KUKA KRL program: EPS_2_251245_SANMH2A_A_20250910012814.src

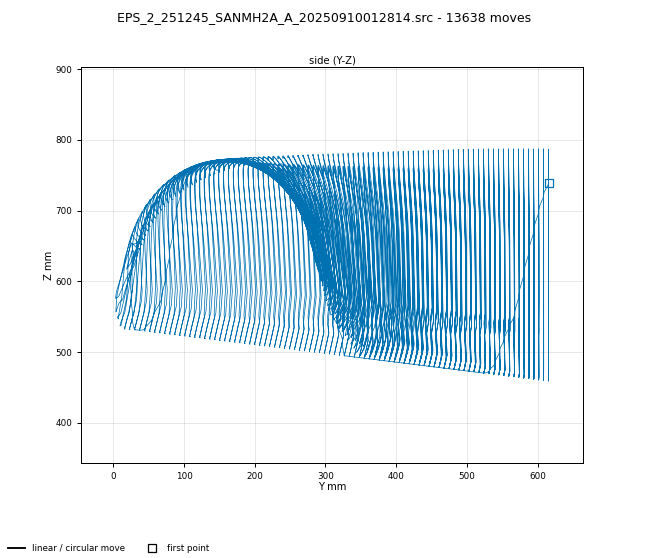
[picture p0: tool path of EPS_2_251245_SANMH2A_A_20250910012814.src, 13638 of 13640 moves have a stored position in this frame; points joined in program order, loops and branches not executed]
&ACCESS RVP
&REL 4
&COMMENT QRS 19112012
&PARAM EDITMASK = *
DEF PART()
EXT BAS (BAS_COMMAND :IN,REAL :IN )
INT I
BAS (#INITMOV,0 )

;KUKA QRS Post kuka4.cps  Date:22-06-2017 !

File_ID=2819

QRS_PRE_INIT()

;Init var - Until changes are made in qrs_pre_init
Outlet_Square_prg=0
Inlet_1_Square_prg=0
Inlet_2_Square_prg=0
Inlet_3_Square_prg=0
Inlet_4_Square_prg=0
Inlet_5_Square_prg=0

Outlet_1={X 0.000, Y 516.340, Z 662.000, B 0.000, E1 0.000 }
Inlet_1={X 0.000, Y 521.550, Z 654.000, B 0.000, E1 91.000 }
Inlet_2={X 0.000, Y 521.330, Z 657.000, B 0.000, E1 270.000 }
Outlet_1_type=251
Inlet_1_type=201
Inlet_2_type=201
;QRS#1=Sidecore dimensions
;QRS#2=250-10" PVC SDR 35
;QRS#3=200-8" PVC SDR 35
;QRS#4=200-8" PVC SDR 35
;QRS#5=
;QRS#6=
;QRS#7=
;QRS#8=
;QRS#9=14M PSX
;QRS#10=12-08 PSX
;QRS#11=12-08 PSX
;QRS#12=
;QRS#13=
;QRS#14=
;QRS#15=
;QRS#16=1220x127x1067 3,5'
;QRS#17=EPS Height
;QRS#18=787,5
;QRS#19=*
;QRS#20= UPDATED VERSION 22-06-2017
;QRS#21=*
Outlet_Square=0100
Inlet_1_Square=0100
Inlet_2_Square=0100
Inlet_3_Square=0
Inlet_4_Square=0
Inlet_5_Square=0
Mill_Square=1
Outlet_Square_Prg=205
Inlet_1_Square_prg=204
Inlet_2_Square_prg=204

QRS_INIT()

$ADVANCE=5

; T1
PTP {E1 173.419,E2 173.419}
PTP {X 0,Y 615.495,A -85,B 0,C 180,E1 173.419,E2 173.419,E3 0,E4 0,E5 0,E6 0}
QRS_SPEED_INIT()
LIN {X 0,Y 615.495,Z 739.089,A -85,B 0,C 180,E1 173.419,E2 173.419,E3 0,E4 0,E5 0,E6 0} C_VEL
LIN {X 0,Y 615.496,Z 732.969,A -85,B 0,C 180,E1 172.455,E2 172.455} C_VEL
LIN {X 0,Y 615.497,Z 725.117,A -85,B 0,C 180,E1 171.464,E2 171.464} C_VEL
LIN {X 0,Y 615.498,Z 715.327,A -85,B 0,C 180,E1 170.47,E2 170.47} C_VEL
LIN {X 0,Y 615.498,Z 705.048,A -85,B 0,C 180,E1 169.64,E2 169.64} C_VEL
LIN {X 0,Y 615.477,Z 693.364,A -85,B 0,C 180,E1 168.885,E2 168.885} C_VEL
LIN {X 0,Y 615.498,Z 681.888,A -85,B 0,C 180,E1 168.306,E2 168.306} C_VEL
LIN {X 0,Y 615.478,Z 669.89,A -85,B 0,C 180,E1 167.846,E2 167.846} C_VEL
LIN {X 0,Y 615.488,Z 657.742,A -85,B 0,C 180,E1 167.512,E2 167.512} C_VEL
LIN {X 0,Y 615.488,Z 644.369,A -85,B 0,C 180,E1 167.281,E2 167.281} C_VEL
LIN {X 0,Y 615.476,Z 541.661,A -85,B 0,C 180,E1 166.073,E2 166.073} C_VEL
LIN {X 0,Y 615.487,Z 518.802,A -85,B 0,C 180,E1 163.243,E2 163.243} C_VEL
LIN {X 0,Y 615.488,Z 495.468,A -85,B 0,C 180,E1 160.315,E2 160.315} C_VEL
LIN {X 0,Y 615.499,Z 472.639,A -85,B 0,C 180,E1 157.405,E2 157.405} C_VEL
LIN {X 0,Y 615.483,Z 458.809,A -85,B 0,C 180,E1 155.593,E2 155.593} C_VEL
LIN {X 0,Y 615.477,Z 458.815,A -85,B 0,C 180,E1 152.822,E2 152.822} C_VEL
LIN {X 0,Y 615.488,Z 458.822,A -85,B 0,C 180,E1 150.206,E2 150.206} C_VEL
LIN {X 0,Y 615.484,Z 458.808,A -85,B 0,C 180,E1 147.542,E2 147.542} C_VEL
LIN {X 0,Y 615.49,Z 458.807,A -85,B 0,C 180,E1 145.185,E2 145.185} C_VEL
LIN {X 0,Y 615.476,Z 458.818,A -85,B 0,C 180,E1 142.757,E2 142.757} C_VEL
LIN {X 0,Y 615.478,Z 458.815,A -85,B 0,C 180,E1 139.912,E2 139.912} C_VEL
LIN {X 0,Y 615.478,Z 458.81,A -85,B 0,C 180,E1 137.646,E2 137.646} C_VEL
LIN {X 0,Y 615.48,Z 458.814,A -85,B 0,C 180,E1 134.931,E2 134.931} C_VEL
LIN {X 0,Y 615.488,Z 458.816,A -85,B 0,C 180,E1 132.08,E2 132.08} C_VEL
LIN {X 0,Y 615.477,Z 458.812,A -85,B 0,C 180,E1 129.751,E2 129.751} C_VEL
LIN {X 0,Y 615.483,Z 458.813,A -85,B 0,C 180,E1 126.936,E2 126.936} C_VEL
LIN {X 0,Y 615.487,Z 458.814,A -85,B 0,C 180,E1 124.022,E2 124.022} C_VEL
LIN {X 0,Y 615.477,Z 458.81,A -85,B 0,C 180,E1 121.686,E2 121.686} C_VEL
LIN {X 0,Y 615.478,Z 458.809,A -85,B 0,C 180,E1 119.407,E2 119.407} C_VEL
LIN {X 0,Y 615.491,Z 458.81,A -85,B 0,C 180,E1 117.046,E2 117.046} C_VEL
LIN {X 0,Y 615.497,Z 458.818,A -85,B 0,C 180,E1 114.272,E2 114.272} C_VEL
LIN {X 0,Y 615.48,Z 458.809,A -85,B 0,C 180,E1 111.432,E2 111.432} C_VEL
LIN {X 0,Y 615.495,Z 458.822,A -85,B 0,C 180,E1 108.607,E2 108.607} C_VEL
LIN {X 0,Y 615.486,Z 458.811,A -85,B 0,C 180,E1 105.905,E2 105.905} C_VEL
LIN {X 0,Y 615.488,Z 458.809,A -85,B 0,C 180,E1 103.201,E2 103.201} C_VEL
LIN {X 0,Y 615.494,Z 458.826,A -85,B 0,C 180,E1 100.527,E2 100.527} C_VEL
LIN {X 0,Y 615.487,Z 458.81,A -85,B 0,C 180,E1 97.876,E2 97.876} C_VEL
LIN {X 0,Y 615.479,Z 458.811,A -85,B 0,C 180,E1 95.241,E2 95.241} C_VEL
LIN {X 0,Y 615.497,Z 458.823,A -85,B 0,C 180,E1 92.618,E2 92.618} C_VEL
LIN {X 0,Y 615.489,Z 458.811,A -85,B 0,C 180,E1 90,E2 90} C_VEL
LIN {X 0,Y 615.478,Z 458.81,A -85,B 0,C 180,E1 87.382,E2 87.382} C_VEL
LIN {X 0,Y 615.495,Z 458.819,A -85,B 0,C 180,E1 84.759,E2 84.759} C_VEL
LIN {X 0,Y 615.493,Z 458.812,A -85,B 0,C 180,E1 82.124,E2 82.124} C_VEL
LIN {X 0,Y 615.476,Z 458.81,A -85,B 0,C 180,E1 79.473,E2 79.473} C_VEL
LIN {X 0,Y 615.496,Z 458.818,A -85,B 0,C 180,E1 76.799,E2 76.799} C_VEL
LIN {X 0,Y 615.491,Z 458.811,A -85,B 0,C 180,E1 74.095,E2 74.095} C_VEL
LIN {X 0,Y 615.477,Z 458.811,A -85,B 0,C 180,E1 71.354,E2 71.354} C_VEL
LIN {X 0,Y 615.496,Z 458.824,A -85,B 0,C 180,E1 68.568,E2 68.568} C_VEL
LIN {X 0,Y 615.487,Z 458.807,A -85,B 0,C 180,E1 65.728,E2 65.728} C_VEL
LIN {X 0,Y 615.492,Z 458.82,A -85,B 0,C 180,E1 62.823,E2 62.823} C_VEL
LIN {X 0,Y 615.499,Z 458.805,A -85,B 0,C 180,E1 59.84,E2 59.84} C_VEL
LIN {X 0,Y 615.481,Z 458.809,A -85,B 0,C 180,E1 57.542,E2 57.542} C_VEL
LIN {X 0,Y 615.478,Z 458.814,A -85,B 0,C 180,E1 55.184,E2 55.184} C_VEL
LIN {X 0,Y 615.494,Z 458.823,A -85,B 0,C 180,E1 52.758,E2 52.758} C_VEL
LIN {X 0,Y 615.491,Z 458.807,A -85,B 0,C 180,E1 49.911,E2 49.911} C_VEL
LIN {X 0,Y 615.49,Z 458.806,A -85,B 0,C 180,E1 47.647,E2 47.647} C_VEL
LIN {X 0,Y 615.481,Z 458.821,A -85,B 0,C 180,E1 44.931,E2 44.931} C_VEL
LIN {X 0,Y 615.478,Z 458.812,A -85,B 0,C 180,E1 42.079,E2 42.079} C_VEL
LIN {X 0,Y 615.498,Z 458.805,A -85,B 0,C 180,E1 39.749,E2 39.749} C_VEL
LIN {X 0,Y 615.478,Z 458.822,A -85,B 0,C 180,E1 36.935,E2 36.935} C_VEL
LIN {X 0,Y 615.491,Z 458.826,A -85,B 0,C 180,E1 34.701,E2 34.701} C_VEL
LIN {X 0,Y 615.479,Z 458.816,A -85,B 0,C 180,E1 32.329,E2 32.329} C_VEL
LIN {X 0,Y 615.488,Z 458.807,A -85,B 0,C 180,E1 29.794,E2 29.794} C_VEL
LIN {X 0,Y 615.482,Z 458.819,A -85,B 0,C 180,E1 27.043,E2 27.043} C_VEL
LIN {X 0,Y 615.478,Z 458.815,A -85,B 0,C 180,E1 24.272,E2 24.272} C_VEL
LIN {X 0,Y 615.486,Z 458.917,A -85,B 0,C 180,E1 23.49,E2 23.49} C_VEL
LIN {X 0,Y 615.485,Z 480.604,A -85,B 0,C 180,E1 20.731,E2 20.731} C_VEL
LIN {X 0,Y 615.49,Z 502.793,A -85,B 0,C 180,E1 17.957,E2 17.957} C_VEL
LIN {X 0,Y 615.491,Z 524.956,A -85,B 0,C 180,E1 15.226,E2 15.226} C_VEL
LIN {X 0,Y 615.481,Z 544.498,A -85,B 0,C 180,E1 12.845,E2 12.845} C_VEL
LIN {X 0,Y 615.489,Z 653.144,A -85,B 0,C 180,E1 11.548,E2 11.548} C_VEL
LIN {X 0,Y 615.484,Z 665.724,A -85,B 0,C 180,E1 11.277,E2 11.277} C_VEL
LIN {X 0,Y 615.49,Z 679.129,A -85,B 0,C 180,E1 10.841,E2 10.841} C_VEL
LIN {X 0,Y 615.481,Z 691.697,A -85,B 0,C 180,E1 10.278,E2 10.278} C_VEL
LIN {X 0,Y 615.493,Z 703.076,A -85,B 0,C 180,E1 9.613,E2 9.613} C_VEL
LIN {X 0,Y 615.498,Z 713.323,A -85,B 0,C 180,E1 8.867,E2 8.867} C_VEL
LIN {X 0,Y 615.498,Z 722.534,A -85,B 0,C 180,E1 8.041,E2 8.041} C_VEL
LIN {X 0,Y 615.499,Z 731.392,A -85,B 0,C 180,E1 7.057,E2 7.057} C_VEL
LIN {X 0,Y 615.497,Z 738.623,A -85,B 0,C 180,E1 6.063,E2 6.063} C_VEL
LIN {X 0,Y 615.497,Z 743.458,A -85,B 0,C 180,E1 5.241,E2 5.241} C_VEL
LIN {X 0,Y 615.493,Z 748.158,A -85,B 0,C 180,E1 4.256,E2 4.256} C_VEL
LIN {X 0,Y 615.495,Z 751.754,A -85,B 0,C 180,E1 3.273,E2 3.273} C_VEL
LIN {X 0,Y 615.496,Z 753.615,A -85,B 0,C 180,E1 2.618,E2 2.618} C_VEL
LIN {X 0,Y 615.497,Z 755.034,A -85,B 0,C 180,E1 1.963,E2 1.963} C_VEL
LIN {X 0,Y 615.496,Z 756.642,A -85,B 0,C 180,E1 0.654,E2 0.654} C_VEL
LIN {X 0,Y 615.494,Z 756.884,A -85,B 0,C 180,E1 0,E2 0} C_VEL
LIN {X 0,Y 615.496,Z 756.705,A -85,B 0,C 180,E1 -0.654,E2 -0.654} C_VEL
LIN {X 0,Y 615.496,Z 755.183,A -85,B 0,C 180,E1 -1.963,E2 -1.963} C_VEL
LIN {X 0,Y 615.498,Z 753.841,A -85,B 0,C 180,E1 -2.618,E2 -2.618} C_VEL
LIN {X 0,Y 615.496,Z 750.994,A -85,B 0,C 180,E1 -3.601,E2 -3.601} C_VEL
LIN {X 0,Y 615.499,Z 747.134,A -85,B 0,C 180,E1 -4.584,E2 -4.584} C_VEL
LIN {X 0,Y 615.498,Z 742.151,A -85,B 0,C 180,E1 -5.57,E2 -5.57} C_VEL
LIN {X 0,Y 615.497,Z 735.701,A -85,B 0,C 180,E1 -6.583,E2 -6.583} C_VEL
LIN {X 0,Y 615.497,Z 728.036,A -85,B 0,C 180,E1 -7.545,E2 -7.545} C_VEL
LIN {X 0,Y 615.498,Z 718.258,A -85,B 0,C 180,E1 -8.537,E2 -8.537} C_VEL
LIN {X 0,Y 615.497,Z 707.993,A -85,B 0,C 180,E1 -9.364,E2 -9.364} C_VEL
LIN {X 0,Y 615.476,Z 696.432,A -85,B 0,C 180,E1 -10.112,E2 -10.112} C_VEL
LIN {X 0,Y 615.497,Z 684.578,A -85,B 0,C 180,E1 -10.707,E2 -10.707} C_VEL
LIN {X 0,Y 615.478,Z 671.66,A -85,B 0,C 180,E1 -11.193,E2 -11.193} C_VEL
LIN {X 0,Y 615.486,Z 659.058,A -85,B 0,C 180,E1 -11.527,E2 -11.527} C_VEL
LIN {X 0,Y 615.487,Z 645.933,A -85,B 0,C 180,E1 -11.736,E2 -11.736} C_VEL
LIN {X 0,Y 615.478,Z 544.549,A -85,B 0,C 180,E1 -12.929,E2 -12.929} C_VEL
LIN {X 0,Y 615.488,Z 521.533,A -85,B 0,C 180,E1 -15.735,E2 -15.735} C_VEL
LIN {X 0,Y 615.491,Z 497.97,A -85,B 0,C 180,E1 -18.646,E2 -18.646} C_VEL
LIN {X 0,Y 615.497,Z 475.763,A -85,B 0,C 180,E1 -21.432,E2 -21.432} C_VEL
LIN {X 0,Y 615.486,Z 458.809,A -85,B 0,C 180,E1 -23.612,E2 -23.612} C_VEL
LIN {X 0,Y 615.48,Z 458.818,A -85,B 0,C 180,E1 -26.445,E2 -26.445} C_VEL
LIN {X 0,Y 615.49,Z 458.823,A -85,B 0,C 180,E1 -28.658,E2 -28.658} C_VEL
LIN {X 0,Y 615.477,Z 458.818,A -85,B 0,C 180,E1 -31.084,E2 -31.084} C_VEL
LIN {X 0,Y 615.485,Z 458.808,A -85,B 0,C 180,E1 -33.533,E2 -33.533} C_VEL
LIN {X 0,Y 615.484,Z 458.82,A -85,B 0,C 180,E1 -36.425,E2 -36.425} C_VEL
LIN {X 0,Y 615.479,Z 458.816,A -85,B 0,C 180,E1 -39.061,E2 -39.061} C_VEL
LIN {X 0,Y 615.482,Z 458.809,A -85,B 0,C 180,E1 -41.474,E2 -41.474} C_VEL
LIN {X 0,Y 615.479,Z 458.817,A -85,B 0,C 180,E1 -44.15,E2 -44.15} C_VEL
LIN {X 0,Y 615.485,Z 458.814,A -85,B 0,C 180,E1 -46.953,E2 -46.953} C_VEL
LIN {X 0,Y 615.478,Z 458.81,A -85,B 0,C 180,E1 -49.393,E2 -49.393} C_VEL
LIN {X 0,Y 615.492,Z 458.813,A -85,B 0,C 180,E1 -51.988,E2 -51.988} C_VEL
LIN {X 0,Y 615.497,Z 458.825,A -85,B 0,C 180,E1 -54.385,E2 -54.385} C_VEL
LIN {X 0,Y 615.49,Z 458.814,A -85,B 0,C 180,E1 -56.764,E2 -56.764} C_VEL
LIN {X 0,Y 615.478,Z 458.811,A -85,B 0,C 180,E1 -59.08,E2 -59.08} C_VEL
LIN {X 0,Y 615.481,Z 458.81,A -85,B 0,C 180,E1 -61.551,E2 -61.551} C_VEL
LIN {X 0,Y 615.493,Z 458.82,A -85,B 0,C 180,E1 -64.43,E2 -64.43} C_VEL
LIN {X 0,Y 615.48,Z 458.809,A -85,B 0,C 180,E1 -67.155,E2 -67.155} C_VEL
LIN {X 0,Y 615.475,Z 458.897,A -85,B 0,C 180,E1 -67.374,E2 -67.374} C_VEL
LIN {X 0,Y 615.496,Z 484.108,A -85,B 0,C 180,E1 -70.141,E2 -70.141} C_VEL
LIN {X 0,Y 615.495,Z 511.278,A -85,B 0,C 180,E1 -73.072,E2 -73.072} C_VEL
LIN {X 0,Y 615.488,Z 523.651,A -85,B 0,C 180,E1 -74.392,E2 -74.392} C_VEL
LIN {X 0,Y 615.485,Z 662.162,A -85,B 0,C 180,E1 -76.05,E2 -76.05} C_VEL
LIN {X 0,Y 615.486,Z 675.855,A -85,B 0,C 180,E1 -76.336,E2 -76.336} C_VEL
LIN {X 0,Y 615.496,Z 689.566,A -85,B 0,C 180,E1 -76.757,E2 -76.757} C_VEL
LIN {X 0,Y 615.497,Z 702.836,A -85,B 0,C 180,E1 -77.302,E2 -77.302} C_VEL
LIN {X 0,Y 615.492,Z 715.599,A -85,B 0,C 180,E1 -77.972,E2 -77.972} C_VEL
LIN {X 0,Y 615.499,Z 727.182,A -85,B 0,C 180,E1 -78.724,E2 -78.724} C_VEL
LIN {X 0,Y 615.498,Z 738.748,A -85,B 0,C 180,E1 -79.64,E2 -79.64} C_VEL
LIN {X 0,Y 615.497,Z 749.088,A -85,B 0,C 180,E1 -80.636,E2 -80.636} C_VEL
LIN {X 0,Y 615.497,Z 757.602,A -85,B 0,C 180,E1 -81.629,E2 -81.629} C_VEL
LIN {X 0,Y 615.496,Z 765.726,A -85,B 0,C 180,E1 -82.784,E2 -82.784} C_VEL
LIN {X 0,Y 615.496,Z 771.43,A -85,B 0,C 180,E1 -83.773,E2 -83.773} C_VEL
LIN {X 0,Y 615.495,Z 776.08,A -85,B 0,C 180,E1 -84.759,E2 -84.759} C_VEL
LIN {X 0,Y 615.494,Z 780.902,A -85,B 0,C 180,E1 -86.072,E2 -86.072} C_VEL
LIN {X 0,Y 615.496,Z 784.252,A -85,B 0,C 180,E1 -87.382,E2 -87.382} C_VEL
LIN {X 0,Y 615.489,Z 786.229,A -85,B 0,C 180,E1 -88.691,E2 -88.691} C_VEL
LIN {X 0,Y 615.493,Z 786.889,A -85,B 0,C 180,E1 -90,E2 -90} C_VEL
LIN {X 0,Y 615.489,Z 786.229,A -85,B 0,C 180,E1 -91.309,E2 -91.309} C_VEL
LIN {X 0,Y 615.496,Z 784.252,A -85,B 0,C 180,E1 -92.618,E2 -92.618} C_VEL
LIN {X 0,Y 615.494,Z 780.901,A -85,B 0,C 180,E1 -93.929,E2 -93.929} C_VEL
LIN {X 0,Y 615.495,Z 776.08,A -85,B 0,C 180,E1 -95.241,E2 -95.241} C_VEL
LIN {X 0,Y 615.495,Z 769.628,A -85,B 0,C 180,E1 -96.557,E2 -96.557} C_VEL
LIN {X 0,Y 615.497,Z 762.44,A -85,B 0,C 180,E1 -97.711,E2 -97.711} C_VEL
LIN {X 0,Y 615.497,Z 754.902,A -85,B 0,C 180,E1 -98.702,E2 -98.702} C_VEL
LIN {X 0,Y 615.495,Z 745.852,A -85,B 0,C 180,E1 -99.696,E2 -99.696} C_VEL
LIN {X 0,Y 615.497,Z 735.756,A -85,B 0,C 180,E1 -100.618,E2 -100.618} C_VEL
LIN {X 0,Y 615.498,Z 724.855,A -85,B 0,C 180,E1 -101.443,E2 -101.443} C_VEL
LIN {X 0,Y 615.488,Z 712.703,A -85,B 0,C 180,E1 -102.195,E2 -102.195} C_VEL
LIN {X 0,Y 615.495,Z 699.087,A -85,B 0,C 180,E1 -102.865,E2 -102.865} C_VEL
LIN {X 0,Y 615.492,Z 685.829,A -85,B 0,C 180,E1 -103.369,E2 -103.369} C_VEL
LIN {X 0,Y 615.484,Z 672.279,A -85,B 0,C 180,E1 -103.748,E2 -103.748} C_VEL
LIN {X 0,Y 615.486,Z 658.082,A -85,B 0,C 180,E1 -104.008,E2 -104.008} C_VEL
LIN {X 0,Y 615.488,Z 523.65,A -85,B 0,C 180,E1 -105.608,E2 -105.608} C_VEL
LIN {X 0,Y 615.488,Z 497.182,A -85,B 0,C 180,E1 -108.443,E2 -108.443} C_VEL
LIN {X 0,Y 615.493,Z 471.313,A -85,B 0,C 180,E1 -111.256,E2 -111.256} C_VEL
LIN {X 0,Y 615.475,Z 458.811,A -85,B 0,C 180,E1 -112.657,E2 -112.657} C_VEL
LIN {X 0,Y 615.488,Z 458.809,A -85,B 0,C 180,E1 -114.992,E2 -114.992} C_VEL
LIN {X 0,Y 615.492,Z 458.817,A -85,B 0,C 180,E1 -117.915,E2 -117.915} C_VEL
LIN {X 0,Y 615.499,Z 458.808,A -85,B 0,C 180,E1 -120.16,E2 -120.16} C_VEL
LIN {X 0,Y 615.481,Z 458.809,A -85,B 0,C 180,E1 -122.458,E2 -122.458} C_VEL
LIN {X 0,Y 615.478,Z 458.813,A -85,B 0,C 180,E1 -124.816,E2 -124.816} C_VEL
LIN {X 0,Y 615.492,Z 458.823,A -85,B 0,C 180,E1 -127.242,E2 -127.242} C_VEL
LIN {X 0,Y 615.489,Z 458.808,A -85,B 0,C 180,E1 -130.089,E2 -130.089} C_VEL
LIN {X 0,Y 615.486,Z 458.823,A -85,B 0,C 180,E1 -133.047,E2 -133.047} C_VEL
LIN {X 0,Y 615.482,Z 458.809,A -85,B 0,C 180,E1 -136.003,E2 -136.003} C_VEL
LIN {X 0,Y 615.49,Z 458.823,A -85,B 0,C 180,E1 -138.906,E2 -138.906} C_VEL
LIN {X 0,Y 615.496,Z 458.82,A -85,B 0,C 180,E1 -141.096,E2 -141.096} C_VEL
LIN {X 0,Y 615.481,Z 458.811,A -85,B 0,C 180,E1 -143.575,E2 -143.575} C_VEL
LIN {X 0,Y 615.479,Z 458.81,A -85,B 0,C 180,E1 -145.977,E2 -145.977} C_VEL
LIN {X 0,Y 615.493,Z 458.82,A -85,B 0,C 180,E1 -148.914,E2 -148.914} C_VEL
LIN {X 0,Y 615.484,Z 458.809,A -85,B 0,C 180,E1 -151.551,E2 -151.551} C_VEL
LIN {X 0,Y 615.499,Z 458.821,A -85,B 0,C 180,E1 -154.43,E2 -154.43} C_VEL
LIN {X 0,Y 615.484,Z 458.811,A -85,B 0,C 180,E1 -157.155,E2 -157.155} C_VEL
LIN {X 0,Y 615.479,Z 458.836,A -85,B 0,C 180,E1 -157.708,E2 -157.708} C_VEL
LIN {X 0,Y 615.492,Z 480.389,A -85,B 0,C 180,E1 -160.489,E2 -160.489} C_VEL
LIN {X 0,Y 615.492,Z 503.466,A -85,B 0,C 180,E1 -163.413,E2 -163.413} C_VEL
LIN {X 0,Y 615.485,Z 526.538,A -85,B 0,C 180,E1 -166.294,E2 -166.294} C_VEL
LIN {X 0,Y 615.48,Z 541.632,A -85,B 0,C 180,E1 -168.16,E2 -168.16} C_VEL
LIN {X 0,Y 615.491,Z 651.28,A -85,B 0,C 180,E1 -169.473,E2 -169.473} C_VEL
LIN {X 0,Y 615.484,Z 664.198,A -85,B 0,C 180,E1 -169.764,E2 -169.764} C_VEL
LIN {X 0,Y 615.49,Z 676.689,A -85,B 0,C 180,E1 -170.179,E2 -170.179} C_VEL
LIN {X 0,Y 615.482,Z 688.618,A -85,B 0,C 180,E1 -170.718,E2 -170.718} C_VEL
LIN {X 0,Y 615.494,Z 699.982,A -85,B 0,C 180,E1 -171.381,E2 -171.381} C_VEL
LIN {X 0,Y 615.498,Z 710.219,A -85,B 0,C 180,E1 -172.124,E2 -172.124} C_VEL
LIN {X 0,Y 615.499,Z 719.371,A -85,B 0,C 180,E1 -172.943,E2 -172.943} C_VEL
LIN {X 0,Y 615.496,Z 728.347,A -85,B 0,C 180,E1 -173.937,E2 -173.937} C_VEL
LIN {X 0,Y 615.497,Z 735.529,A -85,B 0,C 180,E1 -174.923,E2 -174.923} C_VEL
LIN {X 0,Y 615.493,Z 740.375,A -85,B 0,C 180,E1 -175.744,E2 -175.744} C_VEL
LIN {X 0,Y 615.496,Z 745.086,A -85,B 0,C 180,E1 -176.727,E2 -176.727} C_VEL
LIN {X 0,Y 615.498,Z 748.698,A -85,B 0,C 180,E1 -177.71,E2 -177.71} C_VEL
LIN {X 0,Y 615.496,Z 751.317,A -85,B 0,C 180,E1 -178.691,E2 -178.691} C_VEL
LIN {X 0,Y 615.495,Z 753.389,A -85,B 0,C 180,E1 -180,E2 -180} C_VEL
LIN {X 0,Y 615.496,Z 753.831,A -85,B 0,C 180,E1 -181.309,E2 -181.309} C_VEL
LIN {X 0,Y 615.495,Z 752.757,A -85,B 0,C 180,E1 -182.618,E2 -182.618} C_VEL
LIN {X 0,Y 615.497,Z 751.59,A -85,B 0,C 180,E1 -183.273,E2 -183.273} C_VEL
LIN {X 0,Y 615.494,Z 750.023,A -85,B 0,C 180,E1 -183.928,E2 -183.928} C_VEL
LIN {X 0,Y 615.494,Z 746.868,A -85,B 0,C 180,E1 -184.913,E2 -184.913} C_VEL
LIN {X 0,Y 615.498,Z 742.661,A -85,B 0,C 180,E1 -185.898,E2 -185.898} C_VEL
LIN {X 0,Y 615.495,Z 739.089,A -85,B 0,C 180,E1 -186.581,E2 -186.581} C_VEL
LIN {X 0,Y 614.823,Z 736.384,A -85,B 0,C 180,E1 -187.059,E2 -187.059} C_VEL
LIN {X 0,Y 611.979,Z 731.579,A -85,B 0,C 180,E1 -187.825,E2 -187.825} C_VEL
LIN {X 0,Y 609.133,Z 726.046,A -85,B 0,C 180,E1 -188.558,E2 -188.558} C_VEL
LIN {X 0,Y 608.473,Z 722.206,A -85,B 0,C 180,E1 -188.982,E2 -188.982} C_VEL
LIN {X 0,Y 608.488,Z 713.552,A -85,B 0,C 180,E1 -189.809,E2 -189.809} C_VEL
LIN {X 0,Y 608.492,Z 702.773,A -85,B 0,C 180,E1 -190.649,E2 -190.649} C_VEL
LIN {X 0,Y 608.481,Z 691.914,A -85,B 0,C 180,E1 -191.324,E2 -191.324} C_VEL
LIN {X 0,Y 608.508,Z 679.767,A -85,B 0,C 180,E1 -191.914,E2 -191.914} C_VEL
LIN {X 0,Y 608.523,Z 667.028,A -85,B 0,C 180,E1 -192.379,E2 -192.379} C_VEL
LIN {X 0,Y 608.553,Z 654.338,A -85,B 0,C 180,E1 -192.696,E2 -192.696} C_VEL
LIN {X 0,Y 608.536,Z 638.078,A -85,B 0,C 180,E1 -192.93,E2 -192.93} C_VEL
LIN {X 0,Y 608.466,Z 541.843,A -85,B 0,C 180,E1 -194.072,E2 -194.072} C_VEL
LIN {X 0,Y 608.495,Z 520.137,A -85,B 0,C 180,E1 -196.783,E2 -196.783} C_VEL
LIN {X 0,Y 608.555,Z 498.132,A -85,B 0,C 180,E1 -199.567,E2 -199.567} C_VEL
LIN {X 0,Y 608.592,Z 475.299,A -85,B 0,C 180,E1 -202.506,E2 -202.506} C_VEL
LIN {X 0,Y 608.482,Z 459.811,A -85,B 0,C 180,E1 -204.538,E2 -204.538} C_VEL
LIN {X 0,Y 608.473,Z 459.814,A -85,B 0,C 180,E1 -207.206,E2 -207.206} C_VEL
LIN {X 0,Y 608.466,Z 459.816,A -85,B 0,C 180,E1 -209.971,E2 -209.971} C_VEL
LIN {X 0,Y 608.452,Z 459.813,A -85,B 0,C 180,E1 -212.88,E2 -212.88} C_VEL
LIN {X 0,Y 608.452,Z 459.817,A -85,B 0,C 180,E1 -215.277,E2 -215.277} C_VEL
LIN {X 0,Y 608.461,Z 459.819,A -85,B 0,C 180,E1 -217.747,E2 -217.747} C_VEL
LIN {X 0,Y 608.446,Z 459.814,A -85,B 0,C 180,E1 -220.328,E2 -220.328} C_VEL
LIN {X 0,Y 608.469,Z 459.816,A -85,B 0,C 180,E1 -223.308,E2 -223.308} C_VEL
LIN {X 0,Y 608.47,Z 459.812,A -85,B 0,C 180,E1 -226.13,E2 -226.13} C_VEL
LIN {X 0,Y 608.453,Z 459.813,A -85,B 0,C 180,E1 -228.823,E2 -228.823} C_VEL
LIN {X 0,Y 608.469,Z 459.817,A -85,B 0,C 180,E1 -231.76,E2 -231.76} C_VEL
LIN {X 0,Y 608.447,Z 459.817,A -85,B 0,C 180,E1 -233.955,E2 -233.955} C_VEL
LIN {X 0,Y 608.449,Z 459.813,A -85,B 0,C 180,E1 -236.328,E2 -236.328} C_VEL
LIN {X 0,Y 608.449,Z 459.813,A -85,B 0,C 180,E1 -238.732,E2 -238.732} C_VEL
LIN {X 0,Y 608.477,Z 459.817,A -85,B 0,C 180,E1 -241.379,E2 -241.379} C_VEL
LIN {X 0,Y 608.444,Z 459.817,A -85,B 0,C 180,E1 -243.964,E2 -243.964} C_VEL
LIN {X 0,Y 608.466,Z 459.812,A -85,B 0,C 180,E1 -246.155,E2 -246.155} C_VEL
LIN {X 0,Y 608.469,Z 459.81,A -85,B 0,C 180,E1 -248.308,E2 -248.308} C_VEL
LIN {X 0,Y 608.477,Z 459.816,A -85,B 0,C 180,E1 -251.283,E2 -251.283} C_VEL
LIN {X 0,Y 608.464,Z 459.815,A -85,B 0,C 180,E1 -253.906,E2 -253.906} C_VEL
LIN {X 0,Y 608.465,Z 459.811,A -85,B 0,C 180,E1 -256.643,E2 -256.643} C_VEL
LIN {X 0,Y 608.472,Z 459.818,A -85,B 0,C 180,E1 -259.35,E2 -259.35} C_VEL
LIN {X 0,Y 608.48,Z 459.811,A -85,B 0,C 180,E1 -262.033,E2 -262.033} C_VEL
LIN {X 0,Y 608.46,Z 459.812,A -85,B 0,C 180,E1 -264.698,E2 -264.698} C_VEL
LIN {X 0,Y 608.487,Z 459.817,A -85,B 0,C 180,E1 -267.352,E2 -267.352} C_VEL
LIN {X 0,Y 608.48,Z 459.811,A -85,B 0,C 180,E1 -270,E2 -270} C_VEL
LIN {X 0,Y 608.47,Z 459.81,A -85,B 0,C 180,E1 -272.648,E2 -272.648} C_VEL
LIN {X 0,Y 608.474,Z 459.818,A -85,B 0,C 180,E1 -275.302,E2 -275.302} C_VEL
LIN {X 0,Y 608.481,Z 459.811,A -85,B 0,C 180,E1 -277.967,E2 -277.967} C_VEL
LIN {X 0,Y 608.458,Z 459.812,A -85,B 0,C 180,E1 -280.65,E2 -280.65} C_VEL
LIN {X 0,Y 608.472,Z 459.82,A -85,B 0,C 180,E1 -283.356,E2 -283.356} C_VEL
LIN {X 0,Y 608.462,Z 459.812,A -85,B 0,C 180,E1 -286.094,E2 -286.094} C_VEL
LIN {X 0,Y 608.455,Z 459.814,A -85,B 0,C 180,E1 -288.87,E2 -288.87} C_VEL
LIN {X 0,Y 608.477,Z 459.814,A -85,B 0,C 180,E1 -291.691,E2 -291.691} C_VEL
LIN {X 0,Y 608.455,Z 459.812,A -85,B 0,C 180,E1 -294.571,E2 -294.571} C_VEL
LIN {X 0,Y 608.485,Z 459.816,A -85,B 0,C 180,E1 -297.208,E2 -297.208} C_VEL
LIN {X 0,Y 608.471,Z 459.811,A -85,B 0,C 180,E1 -299.972,E2 -299.972} C_VEL
LIN {X 0,Y 608.459,Z 459.814,A -85,B 0,C 180,E1 -302.88,E2 -302.88} C_VEL
LIN {X 0,Y 608.44,Z 459.824,A -85,B 0,C 180,E1 -305.278,E2 -305.278} C_VEL
LIN {X 0,Y 608.473,Z 459.813,A -85,B 0,C 180,E1 -307.746,E2 -307.746} C_VEL
LIN {X 0,Y 608.451,Z 459.812,A -85,B 0,C 180,E1 -310.329,E2 -310.329} C_VEL
LIN {X 0,Y 608.486,Z 459.819,A -85,B 0,C 180,E1 -313.31,E2 -313.31} C_VEL
LIN {X 0,Y 608.468,Z 459.81,A -85,B 0,C 180,E1 -316.13,E2 -316.13} C_VEL
LIN {X 0,Y 608.449,Z 459.816,A -85,B 0,C 180,E1 -318.823,E2 -318.823} C_VEL
LIN {X 0,Y 608.466,Z 459.819,A -85,B 0,C 180,E1 -321.412,E2 -321.412} C_VEL
LIN {X 0,Y 608.449,Z 459.814,A -85,B 0,C 180,E1 -323.955,E2 -323.955} C_VEL
LIN {X 0,Y 608.451,Z 459.812,A -85,B 0,C 180,E1 -326.328,E2 -326.328} C_VEL
LIN {X 0,Y 608.447,Z 459.815,A -85,B 0,C 180,E1 -328.733,E2 -328.733} C_VEL
LIN {X 0,Y 608.475,Z 459.818,A -85,B 0,C 180,E1 -331.38,E2 -331.38} C_VEL
LIN {X 0,Y 608.478,Z 459.809,A -85,B 0,C 180,E1 -334.278,E2 -334.278} C_VEL
LIN {X 0,Y 608.504,Z 459.962,A -85,B 0,C 180,E1 -336.36,E2 -336.36} C_VEL
LIN {X 0,Y 608.596,Z 476.445,A -85,B 0,C 180,E1 -338.491,E2 -338.491} C_VEL
LIN {X 0,Y 608.545,Z 498.307,A -85,B 0,C 180,E1 -341.264,E2 -341.264} C_VEL
LIN {X 0,Y 608.519,Z 520.864,A -85,B 0,C 180,E1 -344.08,E2 -344.08} C_VEL
LIN {X 0,Y 608.473,Z 543.075,A -85,B 0,C 180,E1 -346.814,E2 -346.814} C_VEL
LIN {X 0,Y 608.481,Z 544.724,A -85,B 0,C 180,E1 -347.016,E2 -347.016} C_VEL
LIN {X 0,Y 608.554,Z 653.284,A -85,B 0,C 180,E1 -348.319,E2 -348.319} C_VEL
LIN {X 0,Y 608.531,Z 666.622,A -85,B 0,C 180,E1 -348.614,E2 -348.614} C_VEL
LIN {X 0,Y 608.511,Z 679.096,A -85,B 0,C 180,E1 -349.026,E2 -349.026} C_VEL
LIN {X 0,Y 608.509,Z 690.233,A -85,B 0,C 180,E1 -349.519,E2 -349.519} C_VEL
LIN {X 0,Y 608.488,Z 702.014,A -85,B 0,C 180,E1 -350.191,E2 -350.191} C_VEL
LIN {X 0,Y 608.474,Z 713.585,A -85,B 0,C 180,E1 -351.029,E2 -351.029} C_VEL
LIN {X 0,Y 608.464,Z 722.849,A -85,B 0,C 180,E1 -351.866,E2 -351.866} C_VEL
LIN {X 0,Y 608.466,Z 731.823,A -85,B 0,C 180,E1 -352.867,E2 -352.867} C_VEL
LIN {X 0,Y 608.444,Z 739.056,A -85,B 0,C 180,E1 -353.867,E2 -353.867} C_VEL
LIN {X 0,Y 608.462,Z 743.935,A -85,B 0,C 180,E1 -354.698,E2 -354.698} C_VEL
LIN {X 0,Y 608.439,Z 748.679,A -85,B 0,C 180,E1 -355.694,E2 -355.694} C_VEL
LIN {X 0,Y 608.426,Z 752.313,A -85,B 0,C 180,E1 -356.689,E2 -356.689} C_VEL
LIN {X 0,Y 608.425,Z 754.19,A -85,B 0,C 180,E1 -357.352,E2 -357.352} C_VEL
LIN {X 0,Y 608.442,Z 755.626,A -85,B 0,C 180,E1 -358.014,E2 -358.014} C_VEL
LIN {X 0,Y 608.439,Z 757.252,A -85,B 0,C 180,E1 -359.338,E2 -359.338} C_VEL
LIN {X 0,Y 608.434,Z 757.495,A -85,B 0,C 180,E1 -360,E2 -360} C_VEL
LIN {X 0,Y 608.439,Z 757.315,A -85,B 0,C 180,E1 -360.662,E2 -360.662} C_VEL
LIN {X 0,Y 608.441,Z 755.776,A -85,B 0,C 180,E1 -361.986,E2 -361.986} C_VEL
LIN {X 0,Y 608.426,Z 754.419,A -85,B 0,C 180,E1 -362.648,E2 -362.648} C_VEL
LIN {X 0,Y 608.449,Z 751.542,A -85,B 0,C 180,E1 -363.642,E2 -363.642} C_VEL
LIN {X 0,Y 608.433,Z 747.643,A -85,B 0,C 180,E1 -364.638,E2 -364.638} C_VEL
LIN {X 0,Y 608.449,Z 742.613,A -85,B 0,C 180,E1 -365.634,E2 -365.634} C_VEL
LIN {X 0,Y 608.442,Z 736.292,A -85,B 0,C 180,E1 -366.633,E2 -366.633} C_VEL
LIN {X 0,Y 608.475,Z 728.379,A -85,B 0,C 180,E1 -367.633,E2 -367.633} C_VEL
LIN {X 0,Y 608.472,Z 718.536,A -85,B 0,C 180,E1 -368.636,E2 -368.636} C_VEL
LIN {X 0,Y 608.48,Z 708.209,A -85,B 0,C 180,E1 -369.473,E2 -369.473} C_VEL
LIN {X 0,Y 608.473,Z 696.595,A -85,B 0,C 180,E1 -370.229,E2 -370.229} C_VEL
LIN {X 0,Y 608.525,Z 685.402,A -85,B 0,C 180,E1 -370.801,E2 -370.801} C_VEL
LIN {X 0,Y 608.527,Z 672.754,A -85,B 0,C 180,E1 -371.29,E2 -371.29} C_VEL
LIN {X 0,Y 608.53,Z 660.049,A -85,B 0,C 180,E1 -371.639,E2 -371.639} C_VEL
LIN {X 0,Y 608.559,Z 647.787,A -85,B 0,C 180,E1 -371.85,E2 -371.85} C_VEL
LIN {X 0,Y 608.466,Z 544.678,A -85,B 0,C 180,E1 -373.08,E2 -373.08} C_VEL
LIN {X 0,Y 608.497,Z 522.979,A -85,B 0,C 180,E1 -375.749,E2 -375.749} C_VEL
LIN {X 0,Y 608.56,Z 500.92,A -85,B 0,C 180,E1 -378.497,E2 -378.497} C_VEL
LIN {X 0,Y 608.564,Z 479.925,A -85,B 0,C 180,E1 -381.155,E2 -381.155} C_VEL
LIN {X 0,Y 608.6,Z 460.481,A -85,B 0,C 180,E1 -383.659,E2 -383.659} C_VEL
LIN {X 0,Y 608.485,Z 459.81,A -85,B 0,C 180,E1 -383.754,E2 -383.754} C_VEL
LIN {X 0,Y 608.447,Z 459.814,A -85,B 0,C 180,E1 -386.035,E2 -386.035} C_VEL
LIN {X 0,Y 608.473,Z 459.818,A -85,B 0,C 180,E1 -388.619,E2 -388.619} C_VEL
LIN {X 0,Y 608.447,Z 459.815,A -85,B 0,C 180,E1 -391.318,E2 -391.318} C_VEL
LIN {X 0,Y 608.475,Z 459.81,A -85,B 0,C 180,E1 -393.735,E2 -393.735} C_VEL
LIN {X 0,Y 608.449,Z 459.815,A -85,B 0,C 180,E1 -396.092,E2 -396.092} C_VEL
LIN {X 0,Y 608.467,Z 459.821,A -85,B 0,C 180,E1 -398.588,E2 -398.588} C_VEL
LIN {X 0,Y 608.457,Z 459.812,A -85,B 0,C 180,E1 -401.341,E2 -401.341} C_VEL
LIN {X 0,Y 608.45,Z 459.818,A -85,B 0,C 180,E1 -404.263,E2 -404.263} C_VEL
LIN {X 0,Y 608.453,Z 459.815,A -85,B 0,C 180,E1 -407.04,E2 -407.04} C_VEL
LIN {X 0,Y 608.455,Z 459.813,A -85,B 0,C 180,E1 -409.697,E2 -409.697} C_VEL
LIN {X 0,Y 608.476,Z 459.817,A -85,B 0,C 180,E1 -412.254,E2 -412.254} C_VEL
LIN {X 0,Y 608.446,Z 459.818,A -85,B 0,C 180,E1 -414.722,E2 -414.722} C_VEL
LIN {X 0,Y 608.458,Z 459.812,A -85,B 0,C 180,E1 -417.12,E2 -417.12} C_VEL
LIN {X 0,Y 608.473,Z 459.81,A -85,B 0,C 180,E1 -419.455,E2 -419.455} C_VEL
LIN {X 0,Y 608.452,Z 459.815,A -85,B 0,C 180,E1 -421.733,E2 -421.733} C_VEL
LIN {X 0,Y 608.48,Z 459.82,A -85,B 0,C 180,E1 -424.278,E2 -424.278} C_VEL
LIN {X 0,Y 608.478,Z 459.81,A -85,B 0,C 180,E1 -427.147,E2 -427.147} C_VEL
LIN {X 0,Y 608.5,Z 460.122,A -85,B 0,C 180,E1 -427.238,E2 -427.238} C_VEL
LIN {X 0,Y 608.61,Z 477.879,A -85,B 0,C 180,E1 -429.22,E2 -429.22} C_VEL
LIN {X 0,Y 608.546,Z 503.3,A -85,B 0,C 180,E1 -432.005,E2 -432.005} C_VEL
LIN {X 0,Y 608.526,Z 523.691,A -85,B 0,C 180,E1 -434.209,E2 -434.209} C_VEL
LIN {X 0,Y 608.613,Z 662.979,A -85,B 0,C 180,E1 -435.904,E2 -435.904} C_VEL
LIN {X 0,Y 608.583,Z 676.623,A -85,B 0,C 180,E1 -436.2,E2 -436.2} C_VEL
LIN {X 0,Y 608.581,Z 690.709,A -85,B 0,C 180,E1 -436.646,E2 -436.646} C_VEL
LIN {X 0,Y 608.562,Z 702.881,A -85,B 0,C 180,E1 -437.155,E2 -437.155} C_VEL
LIN {X 0,Y 608.515,Z 715.679,A -85,B 0,C 180,E1 -437.832,E2 -437.832} C_VEL
LIN {X 0,Y 608.499,Z 728.47,A -85,B 0,C 180,E1 -438.677,E2 -438.677} C_VEL
LIN {X 0,Y 608.496,Z 738.93,A -85,B 0,C 180,E1 -439.519,E2 -439.519} C_VEL
LIN {X 0,Y 608.479,Z 749.334,A -85,B 0,C 180,E1 -440.527,E2 -440.527} C_VEL
LIN {X 0,Y 608.464,Z 757.914,A -85,B 0,C 180,E1 -441.531,E2 -441.531} C_VEL
LIN {X 0,Y 608.461,Z 766.113,A -85,B 0,C 180,E1 -442.701,E2 -442.701} C_VEL
LIN {X 0,Y 608.443,Z 772.546,A -85,B 0,C 180,E1 -443.831,E2 -443.831} C_VEL
LIN {X 0,Y 608.437,Z 777.962,A -85,B 0,C 180,E1 -445.03,E2 -445.03} C_VEL
LIN {X 0,Y 608.431,Z 781.441,A -85,B 0,C 180,E1 -446.026,E2 -446.026} C_VEL
LIN {X 0,Y 608.424,Z 784.831,A -85,B 0,C 180,E1 -447.352,E2 -447.352} C_VEL
LIN {X 0,Y 608.442,Z 786.83,A -85,B 0,C 180,E1 -448.676,E2 -448.676} C_VEL
LIN {X 0,Y 608.433,Z 787.5,A -85,B 0,C 180,E1 -450,E2 -450} C_VEL
LIN {X 0,Y 608.442,Z 786.83,A -85,B 0,C 180,E1 -451.324,E2 -451.324} C_VEL
LIN {X 0,Y 608.424,Z 784.831,A -85,B 0,C 180,E1 -452.648,E2 -452.648} C_VEL
LIN {X 0,Y 608.431,Z 781.441,A -85,B 0,C 180,E1 -453.974,E2 -453.974} C_VEL
LIN {X 0,Y 608.44,Z 776.567,A -85,B 0,C 180,E1 -455.302,E2 -455.302} C_VEL
LIN {X 0,Y 608.445,Z 770.211,A -85,B 0,C 180,E1 -456.604,E2 -456.604} C_VEL
LIN {X 0,Y 608.453,Z 762.797,A -85,B 0,C 180,E1 -457.8,E2 -457.8} C_VEL
LIN {X 0,Y 608.473,Z 753.822,A -85,B 0,C 180,E1 -458.971,E2 -458.971} C_VEL
LIN {X 0,Y 608.472,Z 744.389,A -85,B 0,C 180,E1 -459.977,E2 -459.977} C_VEL
LIN {X 0,Y 608.506,Z 733.047,A -85,B 0,C 180,E1 -460.973,E2 -460.973} C_VEL
LIN {X 0,Y 608.533,Z 721.145,A -85,B 0,C 180,E1 -461.829,E2 -461.829} C_VEL
LIN {X 0,Y 608.531,Z 708.069,A -85,B 0,C 180,E1 -462.591,E2 -462.591} C_VEL
LIN {X 0,Y 608.562,Z 695.168,A -85,B 0,C 180,E1 -463.184,E2 -463.184} C_VEL
LIN {X 0,Y 608.586,Z 681.175,A -85,B 0,C 180,E1 -463.673,E2 -463.673} C_VEL
LIN {X 0,Y 608.598,Z 667.443,A -85,B 0,C 180,E1 -464.013,E2 -464.013} C_VEL
LIN {X 0,Y 608.626,Z 651.149,A -85,B 0,C 180,E1 -464.258,E2 -464.258} C_VEL
LIN {X 0,Y 608.526,Z 523.691,A -85,B 0,C 180,E1 -465.791,E2 -465.791} C_VEL
LIN {X 0,Y 608.58,Z 497.578,A -85,B 0,C 180,E1 -468.617,E2 -468.617} C_VEL
LIN {X 0,Y 608.621,Z 472.912,A -85,B 0,C 180,E1 -471.33,E2 -471.33} C_VEL
LIN {X 0,Y 608.471,Z 459.921,A -85,B 0,C 180,E1 -472.786,E2 -472.786} C_VEL
LIN {X 0,Y 608.455,Z 459.817,A -85,B 0,C 180,E1 -475.301,E2 -475.301} C_VEL
LIN {X 0,Y 608.455,Z 459.821,A -85,B 0,C 180,E1 -477.518,E2 -477.518} C_VEL
LIN {X 0,Y 608.472,Z 459.814,A -85,B 0,C 180,E1 -479.972,E2 -479.972} C_VEL
LIN {X 0,Y 608.458,Z 459.812,A -85,B 0,C 180,E1 -482.522,E2 -482.522} C_VEL
LIN {X 0,Y 608.443,Z 459.816,A -85,B 0,C 180,E1 -484.905,E2 -484.905} C_VEL
LIN {X 0,Y 608.472,Z 459.814,A -85,B 0,C 180,E1 -487.746,E2 -487.746} C_VEL
LIN {X 0,Y 608.45,Z 459.813,A -85,B 0,C 180,E1 -490.329,E2 -490.329} C_VEL
LIN {X 0,Y 608.485,Z 459.817,A -85,B 0,C 180,E1 -493.31,E2 -493.31} C_VEL
LIN {X 0,Y 608.468,Z 459.811,A -85,B 0,C 180,E1 -496.13,E2 -496.13} C_VEL
LIN {X 0,Y 608.458,Z 459.819,A -85,B 0,C 180,E1 -498.824,E2 -498.824} C_VEL
LIN {X 0,Y 608.473,Z 459.813,A -85,B 0,C 180,E1 -501.412,E2 -501.412} C_VEL
LIN {X 0,Y 608.449,Z 459.813,A -85,B 0,C 180,E1 -503.955,E2 -503.955} C_VEL
LIN {X 0,Y 608.467,Z 459.814,A -85,B 0,C 180,E1 -506.329,E2 -506.329} C_VEL
LIN {X 0,Y 608.483,Z 459.82,A -85,B 0,C 180,E1 -508.728,E2 -508.728} C_VEL
LIN {X 0,Y 608.474,Z 459.811,A -85,B 0,C 180,E1 -511.381,E2 -511.381} C_VEL
LIN {X 0,Y 608.48,Z 459.815,A -85,B 0,C 180,E1 -514.278,E2 -514.278} C_VEL
LIN {X 0,Y 608.452,Z 459.818,A -85,B 0,C 180,E1 -516.876,E2 -516.876} C_VEL
LIN {X 0,Y 608.476,Z 459.841,A -85,B 0,C 180,E1 -517.556,E2 -517.556} C_VEL
LIN {X 0,Y 608.579,Z 476.422,A -85,B 0,C 180,E1 -519.73,E2 -519.73} C_VEL
LIN {X 0,Y 608.533,Z 498.161,A -85,B 0,C 180,E1 -522.526,E2 -522.526} C_VEL
LIN {X 0,Y 608.509,Z 519.92,A -85,B 0,C 180,E1 -525.28,E2 -525.28} C_VEL
LIN {X 0,Y 608.488,Z 542.043,A -85,B 0,C 180,E1 -528.022,E2 -528.022} C_VEL
LIN {X 0,Y 608.549,Z 650.843,A -85,B 0,C 180,E1 -529.329,E2 -529.329} C_VEL
LIN {X 0,Y 608.536,Z 663.997,A -85,B 0,C 180,E1 -529.625,E2 -529.625} C_VEL
LIN {X 0,Y 608.511,Z 676.037,A -85,B 0,C 180,E1 -530.024,E2 -530.024} C_VEL
LIN {X 0,Y 608.511,Z 687.395,A -85,B 0,C 180,E1 -530.527,E2 -530.527} C_VEL
LIN {X 0,Y 608.475,Z 699.103,A -85,B 0,C 180,E1 -531.197,E2 -531.197} C_VEL
LIN {X 0,Y 608.481,Z 709.573,A -85,B 0,C 180,E1 -531.95,E2 -531.95} C_VEL
LIN {X 0,Y 608.462,Z 718.155,A -85,B 0,C 180,E1 -532.701,E2 -532.701} C_VEL
LIN {X 0,Y 608.468,Z 725.743,A -85,B 0,C 180,E1 -533.498,E2 -533.498} C_VEL
LIN {X 0,Y 608.462,Z 733.802,A -85,B 0,C 180,E1 -534.532,E2 -534.532} C_VEL
LIN {X 0,Y 608.439,Z 740.914,A -85,B 0,C 180,E1 -535.694,E2 -535.694} C_VEL
LIN {X 0,Y 608.429,Z 745.656,A -85,B 0,C 180,E1 -536.689,E2 -536.689} C_VEL
LIN {X 0,Y 608.43,Z 749.293,A -85,B 0,C 180,E1 -537.683,E2 -537.683} C_VEL
LIN {X 0,Y 608.448,Z 751.928,A -85,B 0,C 180,E1 -538.676,E2 -538.676} C_VEL
LIN {X 0,Y 608.436,Z 754.006,A -85,B 0,C 180,E1 -540,E2 -540} C_VEL
LIN {X 0,Y 608.449,Z 754.441,A -85,B 0,C 180,E1 -541.324,E2 -541.324} C_VEL
LIN {X 0,Y 608.442,Z 754.088,A -85,B 0,C 180,E1 -541.986,E2 -541.986} C_VEL
LIN {X 0,Y 608.422,Z 753.336,A -85,B 0,C 180,E1 -542.648,E2 -542.648} C_VEL
LIN {X 0,Y 608.425,Z 752.15,A -85,B 0,C 180,E1 -543.311,E2 -543.311} C_VEL
LIN {X 0,Y 608.432,Z 749.616,A -85,B 0,C 180,E1 -544.306,E2 -544.306} C_VEL
LIN {X 0,Y 608.441,Z 746.079,A -85,B 0,C 180,E1 -545.302,E2 -545.302} C_VEL
LIN {X 0,Y 608.452,Z 741.061,A -85,B 0,C 180,E1 -546.369,E2 -546.369} C_VEL
LIN {X 0,Y 608.451,Z 734.42,A -85,B 0,C 180,E1 -547.466,E2 -547.466} C_VEL
LIN {X 0,Y 608.464,Z 726.819,A -85,B 0,C 180,E1 -548.469,E2 -548.469} C_VEL
LIN {X 0,Y 608.473,Z 722.206,A -85,B 0,C 180,E1 -548.982,E2 -548.982} C_VEL
LIN {X 0,Y 607.8,Z 718.267,A -85,B 0,C 180,E1 -549.388,E2 -549.388} C_VEL
LIN {X 0,Y 604.934,Z 711.609,A -85,B 0,C 180,E1 -550.03,E2 -550.03} C_VEL
LIN {X 0,Y 602.094,Z 704.487,A -85,B 0,C 180,E1 -550.629,E2 -550.629} C_VEL
LIN {X 0,Y 601.466,Z 699.762,A -85,B 0,C 180,E1 -550.965,E2 -550.965} C_VEL
LIN {X 0,Y 601.51,Z 688.542,A -85,B 0,C 180,E1 -551.627,E2 -551.627} C_VEL
LIN {X 0,Y 601.556,Z 676.388,A -85,B 0,C 180,E1 -552.182,E2 -552.182} C_VEL
LIN {X 0,Y 601.576,Z 663.593,A -85,B 0,C 180,E1 -552.61,E2 -552.61} C_VEL
LIN {X 0,Y 601.606,Z 650.204,A -85,B 0,C 180,E1 -552.91,E2 -552.91} C_VEL
LIN {X 0,Y 601.592,Z 542.915,A -85,B 0,C 180,E1 -554.21,E2 -554.21} C_VEL
LIN {X 0,Y 601.464,Z 541.675,A -85,B 0,C 180,E1 -554.248,E2 -554.248} C_VEL
LIN {X 0,Y 601.527,Z 518.659,A -85,B 0,C 180,E1 -557.158,E2 -557.158} C_VEL
LIN {X 0,Y 601.585,Z 496.651,A -85,B 0,C 180,E1 -559.981,E2 -559.981} C_VEL
LIN {X 0,Y 601.683,Z 475.999,A -85,B 0,C 180,E1 -562.672,E2 -562.672} C_VEL
LIN {X 0,Y 601.652,Z 461.807,A -85,B 0,C 180,E1 -564.554,E2 -564.554} C_VEL
LIN {X 0,Y 601.434,Z 460.691,A -85,B 0,C 180,E1 -564.72,E2 -564.72} C_VEL
LIN {X 0,Y 601.412,Z 460.696,A -85,B 0,C 180,E1 -567.361,E2 -567.361} C_VEL
LIN {X 0,Y 601.431,Z 460.69,A -85,B 0,C 180,E1 -570.164,E2 -570.164} C_VEL
LIN {X 0,Y 601.42,Z 460.688,A -85,B 0,C 180,E1 -572.715,E2 -572.715} C_VEL
LIN {X 0,Y 601.417,Z 460.691,A -85,B 0,C 180,E1 -575.114,E2 -575.114} C_VEL
LIN {X 0,Y 601.435,Z 460.694,A -85,B 0,C 180,E1 -577.419,E2 -577.419} C_VEL
LIN {X 0,Y 601.414,Z 460.693,A -85,B 0,C 180,E1 -579.995,E2 -579.995} C_VEL
LIN {X 0,Y 601.41,Z 460.689,A -85,B 0,C 180,E1 -582.67,E2 -582.67} C_VEL
LIN {X 0,Y 601.429,Z 460.696,A -85,B 0,C 180,E1 -585.482,E2 -585.482} C_VEL
LIN {X 0,Y 601.425,Z 460.688,A -85,B 0,C 180,E1 -588.407,E2 -588.407} C_VEL
LIN {X 0,Y 601.434,Z 460.697,A -85,B 0,C 180,E1 -591.529,E2 -591.529} C_VEL
LIN {X 0,Y 601.386,Z 460.693,A -85,B 0,C 180,E1 -594.245,E2 -594.245} C_VEL
LIN {X 0,Y 601.42,Z 460.688,A -85,B 0,C 180,E1 -596.686,E2 -596.686} C_VEL
LIN {X 0,Y 601.417,Z 460.691,A -85,B 0,C 180,E1 -599.058,E2 -599.058} C_VEL
LIN {X 0,Y 601.436,Z 460.694,A -85,B 0,C 180,E1 -601.373,E2 -601.373} C_VEL
LIN {X 0,Y 601.405,Z 460.699,A -85,B 0,C 180,E1 -603.636,E2 -603.636} C_VEL
LIN {X 0,Y 601.463,Z 460.688,A -85,B 0,C 180,E1 -605.86,E2 -605.86} C_VEL
LIN {X 0,Y 601.409,Z 460.69,A -85,B 0,C 180,E1 -608.761,E2 -608.761} C_VEL
LIN {X 0,Y 601.426,Z 460.696,A -85,B 0,C 180,E1 -611.608,E2 -611.608} C_VEL
LIN {X 0,Y 601.417,Z 460.689,A -85,B 0,C 180,E1 -614.409,E2 -614.409} C_VEL
LIN {X 0,Y 601.425,Z 460.693,A -85,B 0,C 180,E1 -617.172,E2 -617.172} C_VEL
LIN {X 0,Y 601.435,Z 460.69,A -85,B 0,C 180,E1 -619.905,E2 -619.905} C_VEL
LIN {X 0,Y 601.443,Z 460.685,A -85,B 0,C 180,E1 -622.615,E2 -622.615} C_VEL
LIN {X 0,Y 601.432,Z 460.695,A -85,B 0,C 180,E1 -625.308,E2 -625.308} C_VEL
LIN {X 0,Y 601.435,Z 460.689,A -85,B 0,C 180,E1 -627.991,E2 -627.991} C_VEL
LIN {X 0,Y 601.443,Z 460.686,A -85,B 0,C 180,E1 -630.669,E2 -630.669} C_VEL
LIN {X 0,Y 601.439,Z 460.695,A -85,B 0,C 180,E1 -633.349,E2 -633.349} C_VEL
LIN {X 0,Y 601.436,Z 460.688,A -85,B 0,C 180,E1 -636.037,E2 -636.037} C_VEL
LIN {X 0,Y 601.443,Z 460.687,A -85,B 0,C 180,E1 -638.061,E2 -638.061} C_VEL
LIN {X 0,Y 601.426,Z 460.691,A -85,B 0,C 180,E1 -641.012,E2 -641.012} C_VEL
LIN {X 0,Y 601.425,Z 460.697,A -85,B 0,C 180,E1 -643.516,E2 -643.516} C_VEL
LIN {X 0,Y 601.438,Z 460.686,A -85,B 0,C 180,E1 -646.287,E2 -646.287} C_VEL
LIN {X 0,Y 601.42,Z 460.694,A -85,B 0,C 180,E1 -649.099,E2 -649.099} C_VEL
LIN {X 0,Y 601.415,Z 460.691,A -85,B 0,C 180,E1 -651.959,E2 -651.959} C_VEL
LIN {X 0,Y 601.44,Z 460.686,A -85,B 0,C 180,E1 -654.293,E2 -654.293} C_VEL
LIN {X 0,Y 601.456,Z 460.69,A -85,B 0,C 180,E1 -657.111,E2 -657.111} C_VEL
LIN {X 0,Y 601.42,Z 460.699,A -85,B 0,C 180,E1 -659.393,E2 -659.393} C_VEL
LIN {X 0,Y 601.409,Z 460.694,A -85,B 0,C 180,E1 -661.727,E2 -661.727} C_VEL
LIN {X 0,Y 601.429,Z 460.688,A -85,B 0,C 180,E1 -664.119,E2 -664.119} C_VEL
LIN {X 0,Y 601.439,Z 460.696,A -85,B 0,C 180,E1 -667.382,E2 -667.382} C_VEL
LIN {X 0,Y 601.412,Z 460.69,A -85,B 0,C 180,E1 -669.995,E2 -669.995} C_VEL
LIN {X 0,Y 601.414,Z 460.69,A -85,B 0,C 180,E1 -672.67,E2 -672.67} C_VEL
LIN {X 0,Y 601.427,Z 460.688,A -85,B 0,C 180,E1 -674.535,E2 -674.535} C_VEL
LIN {X 0,Y 601.41,Z 460.698,A -85,B 0,C 180,E1 -677.41,E2 -677.41} C_VEL
LIN {X 0,Y 601.443,Z 460.686,A -85,B 0,C 180,E1 -680.464,E2 -680.464} C_VEL
LIN {X 0,Y 601.4,Z 460.699,A -85,B 0,C 180,E1 -683.417,E2 -683.417} C_VEL
LIN {X 0,Y 601.435,Z 460.687,A -85,B 0,C 180,E1 -686.064,E2 -686.064} C_VEL
LIN {X 0,Y 601.421,Z 460.689,A -85,B 0,C 180,E1 -688.546,E2 -688.546} C_VEL
LIN {X 0,Y 601.435,Z 460.695,A -85,B 0,C 180,E1 -691.373,E2 -691.373} C_VEL
LIN {X 0,Y 601.417,Z 460.689,A -85,B 0,C 180,E1 -694.132,E2 -694.132} C_VEL
LIN {X 0,Y 601.441,Z 460.835,A -85,B 0,C 180,E1 -696.18,E2 -696.18} C_VEL
LIN {X 0,Y 601.735,Z 465.484,A -85,B 0,C 180,E1 -696.803,E2 -696.803} C_VEL
LIN {X 0,Y 601.643,Z 487.554,A -85,B 0,C 180,E1 -699.664,E2 -699.664} C_VEL
LIN {X 0,Y 601.564,Z 509.764,A -85,B 0,C 180,E1 -702.492,E2 -702.492} C_VEL
LIN {X 0,Y 601.5,Z 531.974,A -85,B 0,C 180,E1 -705.278,E2 -705.278} C_VEL
LIN {X 0,Y 601.454,Z 544.728,A -85,B 0,C 180,E1 -706.861,E2 -706.861} C_VEL
LIN {X 0,Y 601.659,Z 575.874,A -85,B 0,C 180,E1 -707.241,E2 -707.241} C_VEL
LIN {X 0,Y 601.626,Z 653.283,A -85,B 0,C 180,E1 -708.183,E2 -708.183} C_VEL
LIN {X 0,Y 601.581,Z 666.65,A -85,B 0,C 180,E1 -708.481,E2 -708.481} C_VEL
LIN {X 0,Y 601.552,Z 679.909,A -85,B 0,C 180,E1 -708.928,E2 -708.928} C_VEL
LIN {X 0,Y 601.507,Z 691.883,A -85,B 0,C 180,E1 -709.481,E2 -709.481} C_VEL
LIN {X 0,Y 601.47,Z 703.303,A -85,B 0,C 180,E1 -710.161,E2 -710.161} C_VEL
LIN {X 0,Y 601.438,Z 713.594,A -85,B 0,C 180,E1 -710.924,E2 -710.924} C_VEL
LIN {X 0,Y 601.411,Z 722.853,A -85,B 0,C 180,E1 -711.77,E2 -711.77} C_VEL
LIN {X 0,Y 601.388,Z 731.828,A -85,B 0,C 180,E1 -712.783,E2 -712.783} C_VEL
LIN {X 0,Y 601.376,Z 738.971,A -85,B 0,C 180,E1 -713.781,E2 -713.781} C_VEL
LIN {X 0,Y 601.372,Z 743.94,A -85,B 0,C 180,E1 -714.635,E2 -714.635} C_VEL
LIN {X 0,Y 601.353,Z 748.683,A -85,B 0,C 180,E1 -715.643,E2 -715.643} C_VEL
LIN {X 0,Y 601.345,Z 752.317,A -85,B 0,C 180,E1 -716.65,E2 -716.65} C_VEL
LIN {X 0,Y 601.324,Z 754.189,A -85,B 0,C 180,E1 -717.32,E2 -717.32} C_VEL
LIN {X 0,Y 601.341,Z 755.623,A -85,B 0,C 180,E1 -717.991,E2 -717.991} C_VEL
LIN {X 0,Y 601.339,Z 757.252,A -85,B 0,C 180,E1 -719.33,E2 -719.33} C_VEL
LIN {X 0,Y 601.335,Z 757.491,A -85,B 0,C 180,E1 -720,E2 -720} C_VEL
LIN {X 0,Y 601.339,Z 757.314,A -85,B 0,C 180,E1 -720.67,E2 -720.67} C_VEL
LIN {X 0,Y 601.34,Z 755.774,A -85,B 0,C 180,E1 -722.009,E2 -722.009} C_VEL
LIN {X 0,Y 601.326,Z 754.417,A -85,B 0,C 180,E1 -722.68,E2 -722.68} C_VEL
LIN {X 0,Y 601.368,Z 751.543,A -85,B 0,C 180,E1 -723.685,E2 -723.685} C_VEL
LIN {X 0,Y 601.337,Z 747.643,A -85,B 0,C 180,E1 -724.693,E2 -724.693} C_VEL
LIN {X 0,Y 601.373,Z 742.612,A -85,B 0,C 180,E1 -725.701,E2 -725.701} C_VEL
LIN {X 0,Y 601.382,Z 736.279,A -85,B 0,C 180,E1 -726.711,E2 -726.711} C_VEL
LIN {X 0,Y 601.396,Z 728.375,A -85,B 0,C 180,E1 -727.723,E2 -727.723} C_VEL
LIN {X 0,Y 601.437,Z 718.531,A -85,B 0,C 180,E1 -728.738,E2 -728.738} C_VEL
LIN {X 0,Y 601.448,Z 708.195,A -85,B 0,C 180,E1 -729.585,E2 -729.585} C_VEL
LIN {X 0,Y 601.467,Z 697.994,A -85,B 0,C 180,E1 -730.265,E2 -730.265} C_VEL
LIN {X 0,Y 601.532,Z 687.013,A -85,B 0,C 180,E1 -730.851,E2 -730.851} C_VEL
LIN {X 0,Y 601.554,Z 675.217,A -85,B 0,C 180,E1 -731.34,E2 -731.34} C_VEL
LIN {X 0,Y 601.573,Z 662.756,A -85,B 0,C 180,E1 -731.712,E2 -731.712} C_VEL
LIN {X 0,Y 601.618,Z 649.257,A -85,B 0,C 180,E1 -731.967,E2 -731.967} C_VEL
LIN {X 0,Y 601.599,Z 545.808,A -85,B 0,C 180,E1 -733.211,E2 -733.211} C_VEL
LIN {X 0,Y 601.463,Z 544.5,A -85,B 0,C 180,E1 -733.257,E2 -733.257} C_VEL
LIN {X 0,Y 601.537,Z 522.975,A -85,B 0,C 180,E1 -735.936,E2 -735.936} C_VEL
LIN {X 0,Y 601.615,Z 501.649,A -85,B 0,C 180,E1 -738.625,E2 -738.625} C_VEL
LIN {X 0,Y 601.666,Z 479.921,A -85,B 0,C 180,E1 -741.409,E2 -741.409} C_VEL
LIN {X 0,Y 601.672,Z 461.865,A -85,B 0,C 180,E1 -743.765,E2 -743.765} C_VEL
LIN {X 0,Y 601.446,Z 460.69,A -85,B 0,C 180,E1 -743.958,E2 -743.958} C_VEL
LIN {X 0,Y 601.403,Z 460.695,A -85,B 0,C 180,E1 -746.364,E2 -746.364} C_VEL
LIN {X 0,Y 601.422,Z 460.69,A -85,B 0,C 180,E1 -749.393,E2 -749.393} C_VEL
LIN {X 0,Y 601.402,Z 460.691,A -85,B 0,C 180,E1 -751.727,E2 -751.727} C_VEL
LIN {X 0,Y 601.432,Z 460.689,A -85,B 0,C 180,E1 -754.118,E2 -754.118} C_VEL
LIN {X 0,Y 601.402,Z 460.701,A -85,B 0,C 180,E1 -756.583,E2 -756.583} C_VEL
LIN {X 0,Y 601.443,Z 460.686,A -85,B 0,C 180,E1 -759.536,E2 -759.536} C_VEL
LIN {X 0,Y 601.409,Z 460.7,A -85,B 0,C 180,E1 -762.59,E2 -762.59} C_VEL
LIN {X 0,Y 601.429,Z 460.687,A -85,B 0,C 180,E1 -765.482,E2 -765.482} C_VEL
LIN {X 0,Y 601.429,Z 460.697,A -85,B 0,C 180,E1 -768.407,E2 -768.407} C_VEL
LIN {X 0,Y 601.436,Z 460.687,A -85,B 0,C 180,E1 -771.529,E2 -771.529} C_VEL
LIN {X 0,Y 601.41,Z 460.698,A -85,B 0,C 180,E1 -774.247,E2 -774.247} C_VEL
LIN {X 0,Y 601.431,Z 460.692,A -85,B 0,C 180,E1 -776.687,E2 -776.687} C_VEL
LIN {X 0,Y 601.433,Z 460.688,A -85,B 0,C 180,E1 -779.059,E2 -779.059} C_VEL
LIN {X 0,Y 601.427,Z 460.688,A -85,B 0,C 180,E1 -781.373,E2 -781.373} C_VEL
LIN {X 0,Y 601.406,Z 460.692,A -85,B 0,C 180,E1 -783.636,E2 -783.636} C_VEL
LIN {X 0,Y 601.423,Z 460.696,A -85,B 0,C 180,E1 -786.59,E2 -786.59} C_VEL
LIN {X 0,Y 601.445,Z 460.781,A -85,B 0,C 180,E1 -787.03,E2 -787.03} C_VEL
LIN {X 0,Y 601.792,Z 465.422,A -85,B 0,C 180,E1 -787.57,E2 -787.57} C_VEL
LIN {X 0,Y 601.698,Z 490.506,A -85,B 0,C 180,E1 -790.378,E2 -790.378} C_VEL
LIN {X 0,Y 601.58,Z 517.345,A -85,B 0,C 180,E1 -793.33,E2 -793.33} C_VEL
LIN {X 0,Y 601.557,Z 523.691,A -85,B 0,C 180,E1 -794.021,E2 -794.021} C_VEL
LIN {X 0,Y 601.833,Z 528.61,A -85,B 0,C 180,E1 -794.094,E2 -794.094} C_VEL
LIN {X 0,Y 601.74,Z 662.894,A -85,B 0,C 180,E1 -795.738,E2 -795.738} C_VEL
LIN {X 0,Y 601.691,Z 677.049,A -85,B 0,C 180,E1 -796.05,E2 -796.05} C_VEL
LIN {X 0,Y 601.667,Z 690.71,A -85,B 0,C 180,E1 -796.49,E2 -796.49} C_VEL
LIN {X 0,Y 601.606,Z 704.632,A -85,B 0,C 180,E1 -797.09,E2 -797.09} C_VEL
LIN {X 0,Y 601.546,Z 717.092,A -85,B 0,C 180,E1 -797.775,E2 -797.775} C_VEL
LIN {X 0,Y 601.504,Z 728.471,A -85,B 0,C 180,E1 -798.543,E2 -798.543} C_VEL
LIN {X 0,Y 601.482,Z 738.931,A -85,B 0,C 180,E1 -799.395,E2 -799.395} C_VEL
LIN {X 0,Y 601.43,Z 749.334,A -85,B 0,C 180,E1 -800.415,E2 -800.415} C_VEL
LIN {X 0,Y 601.407,Z 757.913,A -85,B 0,C 180,E1 -801.431,E2 -801.431} C_VEL
LIN {X 0,Y 601.392,Z 766.114,A -85,B 0,C 180,E1 -802.614,E2 -802.614} C_VEL
LIN {X 0,Y 601.361,Z 771.752,A -85,B 0,C 180,E1 -803.604,E2 -803.604} C_VEL
LIN {X 0,Y 601.355,Z 776.568,A -85,B 0,C 180,E1 -804.635,E2 -804.635} C_VEL
LIN {X 0,Y 601.343,Z 781.442,A -85,B 0,C 180,E1 -805.979,E2 -805.979} C_VEL
LIN {X 0,Y 601.323,Z 784.831,A -85,B 0,C 180,E1 -807.32,E2 -807.32} C_VEL
LIN {X 0,Y 601.342,Z 786.831,A -85,B 0,C 180,E1 -808.661,E2 -808.661} C_VEL
LIN {X 0,Y 601.333,Z 787.5,A -85,B 0,C 180,E1 -810,E2 -810} C_VEL
LIN {X 0,Y 601.342,Z 786.831,A -85,B 0,C 180,E1 -811.339,E2 -811.339} C_VEL
LIN {X 0,Y 601.323,Z 784.831,A -85,B 0,C 180,E1 -812.68,E2 -812.68} C_VEL
LIN {X 0,Y 601.343,Z 781.442,A -85,B 0,C 180,E1 -814.021,E2 -814.021} C_VEL
LIN {X 0,Y 601.355,Z 776.567,A -85,B 0,C 180,E1 -815.365,E2 -815.365} C_VEL
LIN {X 0,Y 601.355,Z 770.051,A -85,B 0,C 180,E1 -816.712,E2 -816.712} C_VEL
LIN {X 0,Y 601.398,Z 762.797,A -85,B 0,C 180,E1 -817.892,E2 -817.892} C_VEL
LIN {X 0,Y 601.43,Z 753.822,A -85,B 0,C 180,E1 -819.077,E2 -819.077} C_VEL
LIN {X 0,Y 601.44,Z 744.39,A -85,B 0,C 180,E1 -820.095,E2 -820.095} C_VEL
LIN {X 0,Y 601.505,Z 733.692,A -85,B 0,C 180,E1 -821.05,E2 -821.05} C_VEL
LIN {X 0,Y 601.543,Z 722.424,A -85,B 0,C 180,E1 -821.883,E2 -821.883} C_VEL
LIN {X 0,Y 601.565,Z 709.641,A -85,B 0,C 180,E1 -822.654,E2 -822.654} C_VEL
LIN {X 0,Y 601.631,Z 697.155,A -85,B 0,C 180,E1 -823.253,E2 -823.253} C_VEL
LIN {X 0,Y 601.665,Z 683.899,A -85,B 0,C 180,E1 -823.747,E2 -823.747} C_VEL
LIN {X 0,Y 601.698,Z 669.538,A -85,B 0,C 180,E1 -824.134,E2 -824.134} C_VEL
LIN {X 0,Y 601.748,Z 655.08,A -85,B 0,C 180,E1 -824.377,E2 -824.377} C_VEL
LIN {X 0,Y 601.742,Z 525.026,A -85,B 0,C 180,E1 -825.952,E2 -825.952} C_VEL
LIN {X 0,Y 601.557,Z 523.691,A -85,B 0,C 180,E1 -825.979,E2 -825.979} C_VEL
LIN {X 0,Y 601.623,Z 500.019,A -85,B 0,C 180,E1 -828.571,E2 -828.571} C_VEL
LIN {X 0,Y 601.733,Z 476.111,A -85,B 0,C 180,E1 -831.227,E2 -831.227} C_VEL
LIN {X 0,Y 601.677,Z 461.879,A -85,B 0,C 180,E1 -832.836,E2 -832.836} C_VEL
LIN {X 0,Y 601.437,Z 460.692,A -85,B 0,C 180,E1 -832.995,E2 -832.995} C_VEL
LIN {X 0,Y 601.44,Z 460.696,A -85,B 0,C 180,E1 -835.617,E2 -835.617} C_VEL
LIN {X 0,Y 601.423,Z 460.695,A -85,B 0,C 180,E1 -837.867,E2 -837.867} C_VEL
LIN {X 0,Y 601.432,Z 460.689,A -85,B 0,C 180,E1 -840.164,E2 -840.164} C_VEL
LIN {X 0,Y 601.421,Z 460.689,A -85,B 0,C 180,E1 -842.715,E2 -842.715} C_VEL
LIN {X 0,Y 601.391,Z 460.698,A -85,B 0,C 180,E1 -845.111,E2 -845.111} C_VEL
LIN {X 0,Y 601.438,Z 460.696,A -85,B 0,C 180,E1 -847.419,E2 -847.419} C_VEL
LIN {X 0,Y 601.404,Z 460.692,A -85,B 0,C 180,E1 -849.996,E2 -849.996} C_VEL
LIN {X 0,Y 601.414,Z 460.692,A -85,B 0,C 180,E1 -852.67,E2 -852.67} C_VEL
LIN {X 0,Y 601.428,Z 460.69,A -85,B 0,C 180,E1 -854.535,E2 -854.535} C_VEL
LIN {X 0,Y 601.412,Z 460.694,A -85,B 0,C 180,E1 -857.41,E2 -857.41} C_VEL
LIN {X 0,Y 601.446,Z 460.688,A -85,B 0,C 180,E1 -860.464,E2 -860.464} C_VEL
LIN {X 0,Y 601.409,Z 460.693,A -85,B 0,C 180,E1 -863.417,E2 -863.417} C_VEL
LIN {X 0,Y 601.436,Z 460.688,A -85,B 0,C 180,E1 -866.064,E2 -866.064} C_VEL
LIN {X 0,Y 601.446,Z 460.693,A -85,B 0,C 180,E1 -868.542,E2 -868.542} C_VEL
LIN {X 0,Y 601.434,Z 460.689,A -85,B 0,C 180,E1 -871.373,E2 -871.373} C_VEL
LIN {X 0,Y 601.405,Z 460.692,A -85,B 0,C 180,E1 -873.636,E2 -873.636} C_VEL
LIN {X 0,Y 601.42,Z 460.699,A -85,B 0,C 180,E1 -876.59,E2 -876.59} C_VEL
LIN {X 0,Y 601.438,Z 460.784,A -85,B 0,C 180,E1 -877.39,E2 -877.39} C_VEL
LIN {X 0,Y 601.705,Z 465.666,A -85,B 0,C 180,E1 -878.052,E2 -878.052} C_VEL
LIN {X 0,Y 601.616,Z 486.034,A -85,B 0,C 180,E1 -880.73,E2 -880.73} C_VEL
LIN {X 0,Y 601.551,Z 508.132,A -85,B 0,C 180,E1 -883.587,E2 -883.587} C_VEL
LIN {X 0,Y 601.505,Z 529.846,A -85,B 0,C 180,E1 -886.352,E2 -886.352} C_VEL
LIN {X 0,Y 601.466,Z 541.802,A -85,B 0,C 180,E1 -887.859,E2 -887.859} C_VEL
LIN {X 0,Y 601.649,Z 566.241,A -85,B 0,C 180,E1 -888.162,E2 -888.162} C_VEL
LIN {X 0,Y 601.605,Z 650.729,A -85,B 0,C 180,E1 -889.189,E2 -889.189} C_VEL
LIN {X 0,Y 601.592,Z 664.439,A -85,B 0,C 180,E1 -889.504,E2 -889.504} C_VEL
LIN {X 0,Y 601.528,Z 676.373,A -85,B 0,C 180,E1 -889.907,E2 -889.907} C_VEL
LIN {X 0,Y 601.513,Z 687.648,A -85,B 0,C 180,E1 -890.416,E2 -890.416} C_VEL
LIN {X 0,Y 601.462,Z 699.293,A -85,B 0,C 180,E1 -891.093,E2 -891.093} C_VEL
LIN {X 0,Y 601.45,Z 709.73,A -85,B 0,C 180,E1 -891.855,E2 -891.855} C_VEL
LIN {X 0,Y 601.412,Z 718.288,A -85,B 0,C 180,E1 -892.615,E2 -892.615} C_VEL
LIN {X 0,Y 601.395,Z 727.352,A -85,B 0,C 180,E1 -893.599,E2 -893.599} C_VEL
LIN {X 0,Y 601.376,Z 735.001,A -85,B 0,C 180,E1 -894.635,E2 -894.635} C_VEL
LIN {X 0,Y 601.356,Z 740.984,A -85,B 0,C 180,E1 -895.643,E2 -895.643} C_VEL
LIN {X 0,Y 601.348,Z 745.708,A -85,B 0,C 180,E1 -896.65,E2 -896.65} C_VEL
LIN {X 0,Y 601.341,Z 749.334,A -85,B 0,C 180,E1 -897.656,E2 -897.656} C_VEL
LIN {X 0,Y 601.348,Z 751.954,A -85,B 0,C 180,E1 -898.661,E2 -898.661} C_VEL
LIN {X 0,Y 601.339,Z 753.185,A -85,B 0,C 180,E1 -899.33,E2 -899.33} C_VEL
LIN {X 0,Y 601.336,Z 754.014,A -85,B 0,C 180,E1 -900,E2 -900} C_VEL
LIN {X 0,Y 601.348,Z 754.438,A -85,B 0,C 180,E1 -901.339,E2 -901.339} C_VEL
LIN {X 0,Y 601.341,Z 754.081,A -85,B 0,C 180,E1 -902.009,E2 -902.009} C_VEL
LIN {X 0,Y 601.321,Z 753.313,A -85,B 0,C 180,E1 -902.68,E2 -902.68} C_VEL
LIN {X 0,Y 601.341,Z 752.123,A -85,B 0,C 180,E1 -903.35,E2 -903.35} C_VEL
LIN {X 0,Y 601.348,Z 749.579,A -85,B 0,C 180,E1 -904.357,E2 -904.357} C_VEL
LIN {X 0,Y 601.356,Z 746.026,A -85,B 0,C 180,E1 -905.365,E2 -905.365} C_VEL
LIN {X 0,Y 601.355,Z 740.22,A -85,B 0,C 180,E1 -906.588,E2 -906.588} C_VEL
LIN {X 0,Y 601.388,Z 733.205,A -85,B 0,C 180,E1 -907.723,E2 -907.723} C_VEL
LIN {X 0,Y 601.407,Z 725.247,A -85,B 0,C 180,E1 -908.738,E2 -908.738} C_VEL
LIN {X 0,Y 601.421,Z 715.336,A -85,B 0,C 180,E1 -909.755,E2 -909.755} C_VEL
LIN {X 0,Y 601.468,Z 704.93,A -85,B 0,C 180,E1 -910.605,E2 -910.605} C_VEL
LIN {X 0,Y 601.466,Z 699.762,A -85,B 0,C 180,E1 -910.965,E2 -910.965} C_VEL
LIN {X 0,Y 600.839,Z 694.917,A -85,B 0,C 180,E1 -911.283,E2 -911.283} C_VEL
LIN {X 0,Y 598.017,Z 686.91,A -85,B 0,C 180,E1 -911.775,E2 -911.775} C_VEL
LIN {X 0,Y 595.251,Z 678.565,A -85,B 0,C 180,E1 -912.212,E2 -912.212} C_VEL
LIN {X 0,Y 594.604,Z 673.192,A -85,B 0,C 180,E1 -912.437,E2 -912.437} C_VEL
LIN {X 0,Y 594.624,Z 659.922,A -85,B 0,C 180,E1 -912.847,E2 -912.847} C_VEL
LIN {X 0,Y 594.656,Z 646.396,A -85,B 0,C 180,E1 -913.107,E2 -913.107} C_VEL
LIN {X 0,Y 594.725,Z 543.803,A -85,B 0,C 180,E1 -914.354,E2 -914.354} C_VEL
LIN {X 0,Y 594.443,Z 541.744,A -85,B 0,C 180,E1 -914.398,E2 -914.398} C_VEL
LIN {X 0,Y 594.551,Z 519.93,A -85,B 0,C 180,E1 -917.189,E2 -917.189} C_VEL
LIN {X 0,Y 594.65,Z 496.546,A -85,B 0,C 180,E1 -920.224,E2 -920.224} C_VEL
LIN {X 0,Y 594.791,Z 475.893,A -85,B 0,C 180,E1 -922.95,E2 -922.95} C_VEL
LIN {X 0,Y 594.798,Z 463.629,A -85,B 0,C 180,E1 -924.595,E2 -924.595} C_VEL
LIN {X 0,Y 594.386,Z 461.571,A -85,B 0,C 180,E1 -924.912,E2 -924.912} C_VEL
LIN {X 0,Y 594.372,Z 461.576,A -85,B 0,C 180,E1 -927.523,E2 -927.523} C_VEL
LIN {X 0,Y 594.389,Z 461.566,A -85,B 0,C 180,E1 -930.328,E2 -930.328} C_VEL
LIN {X 0,Y 594.379,Z 461.567,A -85,B 0,C 180,E1 -932.95,E2 -932.95} C_VEL
LIN {X 0,Y 594.36,Z 461.575,A -85,B 0,C 180,E1 -935.408,E2 -935.408} C_VEL
LIN {X 0,Y 594.382,Z 461.57,A -85,B 0,C 180,E1 -937.941,E2 -937.941} C_VEL
LIN {X 0,Y 594.375,Z 461.566,A -85,B 0,C 180,E1 -940.821,E2 -940.821} C_VEL
LIN {X 0,Y 594.368,Z 461.572,A -85,B 0,C 180,E1 -943.299,E2 -943.299} C_VEL
LIN {X 0,Y 594.386,Z 461.566,A -85,B 0,C 180,E1 -946.159,E2 -946.159} C_VEL
LIN {X 0,Y 594.379,Z 461.569,A -85,B 0,C 180,E1 -949.178,E2 -949.178} C_VEL
LIN {X 0,Y 594.389,Z 461.567,A -85,B 0,C 180,E1 -952.059,E2 -952.059} C_VEL
LIN {X 0,Y 594.352,Z 461.569,A -85,B 0,C 180,E1 -954.677,E2 -954.677} C_VEL
LIN {X 0,Y 594.381,Z 461.568,A -85,B 0,C 180,E1 -957.088,E2 -957.088} C_VEL
LIN {X 0,Y 594.388,Z 461.573,A -85,B 0,C 180,E1 -959.672,E2 -959.672} C_VEL
LIN {X 0,Y 594.377,Z 461.565,A -85,B 0,C 180,E1 -962.539,E2 -962.539} C_VEL
LIN {X 0,Y 594.375,Z 461.567,A -85,B 0,C 180,E1 -964.807,E2 -964.807} C_VEL
LIN {X 0,Y 594.365,Z 461.573,A -85,B 0,C 180,E1 -967.265,E2 -967.265} C_VEL
LIN {X 0,Y 594.379,Z 461.569,A -85,B 0,C 180,E1 -969.946,E2 -969.946} C_VEL
LIN {X 0,Y 594.392,Z 461.565,A -85,B 0,C 180,E1 -972.807,E2 -972.807} C_VEL
LIN {X 0,Y 594.392,Z 461.569,A -85,B 0,C 180,E1 -975.826,E2 -975.826} C_VEL
LIN {X 0,Y 594.397,Z 461.563,A -85,B 0,C 180,E1 -978.404,E2 -978.404} C_VEL
LIN {X 0,Y 594.402,Z 461.568,A -85,B 0,C 180,E1 -981.158,E2 -981.158} C_VEL
LIN {X 0,Y 594.373,Z 461.57,A -85,B 0,C 180,E1 -983.891,E2 -983.891} C_VEL
LIN {X 0,Y 594.379,Z 461.566,A -85,B 0,C 180,E1 -986.611,E2 -986.611} C_VEL
LIN {X 0,Y 594.428,Z 461.568,A -85,B 0,C 180,E1 -989.323,E2 -989.323} C_VEL
LIN {X 0,Y 594.405,Z 461.564,A -85,B 0,C 180,E1 -992.033,E2 -992.033} C_VEL
LIN {X 0,Y 594.389,Z 461.565,A -85,B 0,C 180,E1 -994.748,E2 -994.748} C_VEL
LIN {X 0,Y 594.407,Z 461.572,A -85,B 0,C 180,E1 -997.473,E2 -997.473} C_VEL
LIN {X 0,Y 594.394,Z 461.564,A -85,B 0,C 180,E1 -1000.216,E2 -1000.216} C_VEL
LIN {X 0,Y 594.368,Z 461.57,A -85,B 0,C 180,E1 -1002.983,E2 -1002.983} C_VEL
LIN {X 0,Y 594.373,Z 461.57,A -85,B 0,C 180,E1 -1005.781,E2 -1005.781} C_VEL
LIN {X 0,Y 594.384,Z 461.565,A -85,B 0,C 180,E1 -1008.618,E2 -1008.618} C_VEL
LIN {X 0,Y 594.369,Z 461.575,A -85,B 0,C 180,E1 -1011.503,E2 -1011.503} C_VEL
LIN {X 0,Y 594.391,Z 461.564,A -85,B 0,C 180,E1 -1014.446,E2 -1014.446} C_VEL
LIN {X 0,Y 594.387,Z 461.565,A -85,B 0,C 180,E1 -1016.7,E2 -1016.7} C_VEL
LIN {X 0,Y 594.382,Z 461.569,A -85,B 0,C 180,E1 -1018.999,E2 -1018.999} C_VEL
LIN {X 0,Y 594.386,Z 461.57,A -85,B 0,C 180,E1 -1021.644,E2 -1021.644} C_VEL
LIN {X 0,Y 594.379,Z 461.566,A -85,B 0,C 180,E1 -1024.58,E2 -1024.58} C_VEL
LIN {X 0,Y 594.393,Z 461.569,A -85,B 0,C 180,E1 -1027.609,E2 -1027.609} C_VEL
LIN {X 0,Y 594.371,Z 461.567,A -85,B 0,C 180,E1 -1030.567,E2 -1030.567} C_VEL
LIN {X 0,Y 594.383,Z 461.576,A -85,B 0,C 180,E1 -1033.298,E2 -1033.298} C_VEL
LIN {X 0,Y 594.361,Z 461.568,A -85,B 0,C 180,E1 -1036.161,E2 -1036.161} C_VEL
LIN {X 0,Y 594.379,Z 461.566,A -85,B 0,C 180,E1 -1038.536,E2 -1038.536} C_VEL
LIN {X 0,Y 594.387,Z 461.575,A -85,B 0,C 180,E1 -1041.296,E2 -1041.296} C_VEL
LIN {X 0,Y 594.353,Z 461.572,A -85,B 0,C 180,E1 -1043.756,E2 -1043.756} C_VEL
LIN {X 0,Y 594.379,Z 461.565,A -85,B 0,C 180,E1 -1046.239,E2 -1046.239} C_VEL
LIN {X 0,Y 594.371,Z 461.568,A -85,B 0,C 180,E1 -1048.65,E2 -1048.65} C_VEL
LIN {X 0,Y 594.387,Z 461.571,A -85,B 0,C 180,E1 -1051.042,E2 -1051.042} C_VEL
LIN {X 0,Y 594.391,Z 461.566,A -85,B 0,C 180,E1 -1053.977,E2 -1053.977} C_VEL
LIN {X 0,Y 594.425,Z 461.707,A -85,B 0,C 180,E1 -1055.997,E2 -1055.997} C_VEL
LIN {X 0,Y 594.851,Z 465.35,A -85,B 0,C 180,E1 -1056.5,E2 -1056.5} C_VEL
LIN {X 0,Y 594.727,Z 486.171,A -85,B 0,C 180,E1 -1059.236,E2 -1059.236} C_VEL
LIN {X 0,Y 594.621,Z 508.38,A -85,B 0,C 180,E1 -1062.103,E2 -1062.103} C_VEL
LIN {X 0,Y 594.497,Z 530.591,A -85,B 0,C 180,E1 -1064.925,E2 -1064.925} C_VEL
LIN {X 0,Y 594.447,Z 544.733,A -85,B 0,C 180,E1 -1066.704,E2 -1066.704} C_VEL
LIN {X 0,Y 594.786,Z 550.882,A -85,B 0,C 180,E1 -1066.787,E2 -1066.787} C_VEL
LIN {X 0,Y 594.682,Z 653.273,A -85,B 0,C 180,E1 -1068.043,E2 -1068.043} C_VEL
LIN {X 0,Y 594.622,Z 666.678,A -85,B 0,C 180,E1 -1068.344,E2 -1068.344} C_VEL
LIN {X 0,Y 594.56,Z 678.568,A -85,B 0,C 180,E1 -1068.743,E2 -1068.743} C_VEL
LIN {X 0,Y 594.532,Z 690.229,A -85,B 0,C 180,E1 -1069.27,E2 -1069.27} C_VEL
LIN {X 0,Y 594.47,Z 702.038,A -85,B 0,C 180,E1 -1069.958,E2 -1069.958} C_VEL
LIN {X 0,Y 594.406,Z 713.599,A -85,B 0,C 180,E1 -1070.815,E2 -1070.815} C_VEL
LIN {X 0,Y 594.373,Z 722.849,A -85,B 0,C 180,E1 -1071.672,E2 -1071.672} C_VEL
LIN {X 0,Y 594.317,Z 731.833,A -85,B 0,C 180,E1 -1072.697,E2 -1072.697} C_VEL
LIN {X 0,Y 594.285,Z 738.358,A -85,B 0,C 180,E1 -1073.612,E2 -1073.612} C_VEL
LIN {X 0,Y 594.289,Z 743.945,A -85,B 0,C 180,E1 -1074.571,E2 -1074.571} C_VEL
LIN {X 0,Y 594.27,Z 748.688,A -85,B 0,C 180,E1 -1075.591,E2 -1075.591} C_VEL
LIN {X 0,Y 594.268,Z 752.32,A -85,B 0,C 180,E1 -1076.61,E2 -1076.61} C_VEL
LIN {X 0,Y 594.225,Z 754.188,A -85,B 0,C 180,E1 -1077.288,E2 -1077.288} C_VEL
LIN {X 0,Y 594.24,Z 755.617,A -85,B 0,C 180,E1 -1077.967,E2 -1077.967} C_VEL
LIN {X 0,Y 594.248,Z 756.634,A -85,B 0,C 180,E1 -1078.645,E2 -1078.645} C_VEL
LIN {X 0,Y 594.236,Z 757.484,A -85,B 0,C 180,E1 -1080,E2 -1080} C_VEL
LIN {X 0,Y 594.24,Z 757.314,A -85,B 0,C 180,E1 -1080.678,E2 -1080.678} C_VEL
LIN {X 0,Y 594.248,Z 756.738,A -85,B 0,C 180,E1 -1081.355,E2 -1081.355} C_VEL
LIN {X 0,Y 594.226,Z 754.416,A -85,B 0,C 180,E1 -1082.712,E2 -1082.712} C_VEL
LIN {X 0,Y 594.289,Z 751.543,A -85,B 0,C 180,E1 -1083.729,E2 -1083.729} C_VEL
LIN {X 0,Y 594.242,Z 747.643,A -85,B 0,C 180,E1 -1084.749,E2 -1084.749} C_VEL
LIN {X 0,Y 594.299,Z 742.609,A -85,B 0,C 180,E1 -1085.769,E2 -1085.769} C_VEL
LIN {X 0,Y 594.316,Z 736.266,A -85,B 0,C 180,E1 -1086.791,E2 -1086.791} C_VEL
LIN {X 0,Y 594.346,Z 728.371,A -85,B 0,C 180,E1 -1087.816,E2 -1087.816} C_VEL
LIN {X 0,Y 594.381,Z 718.526,A -85,B 0,C 180,E1 -1088.842,E2 -1088.842} C_VEL
LIN {X 0,Y 594.426,Z 708.182,A -85,B 0,C 180,E1 -1089.699,E2 -1089.699} C_VEL
LIN {X 0,Y 594.481,Z 697.98,A -85,B 0,C 180,E1 -1090.386,E2 -1090.386} C_VEL
LIN {X 0,Y 594.559,Z 686.911,A -85,B 0,C 180,E1 -1090.985,E2 -1090.985} C_VEL
LIN {X 0,Y 594.592,Z 674.205,A -85,B 0,C 180,E1 -1091.508,E2 -1091.508} C_VEL
LIN {X 0,Y 594.649,Z 661.809,A -85,B 0,C 180,E1 -1091.872,E2 -1091.872} C_VEL
LIN {X 0,Y 594.689,Z 649.218,A -85,B 0,C 180,E1 -1092.109,E2 -1092.109} C_VEL
LIN {X 0,Y 594.602,Z 545.762,A -85,B 0,C 180,E1 -1093.369,E2 -1093.369} C_VEL
LIN {X 0,Y 594.448,Z 544.496,A -85,B 0,C 180,E1 -1093.416,E2 -1093.416} C_VEL
LIN {X 0,Y 594.551,Z 522.97,A -85,B 0,C 180,E1 -1096.128,E2 -1096.128} C_VEL
LIN {X 0,Y 594.655,Z 501.41,A -85,B 0,C 180,E1 -1098.881,E2 -1098.881} C_VEL
LIN {X 0,Y 594.773,Z 479.916,A -85,B 0,C 180,E1 -1101.67,E2 -1101.67} C_VEL
LIN {X 0,Y 594.896,Z 464.638,A -85,B 0,C 180,E1 -1103.683,E2 -1103.683} C_VEL
LIN {X 0,Y 594.427,Z 461.566,A -85,B 0,C 180,E1 -1104.117,E2 -1104.117} C_VEL
LIN {X 0,Y 594.384,Z 461.575,A -85,B 0,C 180,E1 -1106.7,E2 -1106.7} C_VEL
LIN {X 0,Y 594.384,Z 461.572,A -85,B 0,C 180,E1 -1108.998,E2 -1108.998} C_VEL
LIN {X 0,Y 594.379,Z 461.566,A -85,B 0,C 180,E1 -1111.642,E2 -1111.642} C_VEL
LIN {X 0,Y 594.385,Z 461.574,A -85,B 0,C 180,E1 -1114.58,E2 -1114.58} C_VEL
LIN {X 0,Y 594.39,Z 461.564,A -85,B 0,C 180,E1 -1117.608,E2 -1117.608} C_VEL
LIN {X 0,Y 594.368,Z 461.577,A -85,B 0,C 180,E1 -1120.567,E2 -1120.567} C_VEL
LIN {X 0,Y 594.367,Z 461.568,A -85,B 0,C 180,E1 -1123.3,E2 -1123.3} C_VEL
LIN {X 0,Y 594.385,Z 461.569,A -85,B 0,C 180,E1 -1126.159,E2 -1126.159} C_VEL
LIN {X 0,Y 594.38,Z 461.567,A -85,B 0,C 180,E1 -1129.178,E2 -1129.178} C_VEL
LIN {X 0,Y 594.391,Z 461.569,A -85,B 0,C 180,E1 -1132.059,E2 -1132.059} C_VEL
LIN {X 0,Y 594.358,Z 461.574,A -85,B 0,C 180,E1 -1134.676,E2 -1134.676} C_VEL
LIN {X 0,Y 594.381,Z 461.566,A -85,B 0,C 180,E1 -1137.088,E2 -1137.088} C_VEL
LIN {X 0,Y 594.404,Z 461.564,A -85,B 0,C 180,E1 -1139.669,E2 -1139.669} C_VEL
LIN {X 0,Y 594.377,Z 461.573,A -85,B 0,C 180,E1 -1142.539,E2 -1142.539} C_VEL
LIN {X 0,Y 594.381,Z 461.569,A -85,B 0,C 180,E1 -1144.807,E2 -1144.807} C_VEL
LIN {X 0,Y 594.412,Z 461.718,A -85,B 0,C 180,E1 -1146.851,E2 -1146.851} C_VEL
LIN {X 0,Y 594.936,Z 465.265,A -85,B 0,C 180,E1 -1147.28,E2 -1147.28} C_VEL
LIN {X 0,Y 594.787,Z 487.307,A -85,B 0,C 180,E1 -1149.78,E2 -1149.78} C_VEL
LIN {X 0,Y 594.675,Z 512.896,A -85,B 0,C 180,E1 -1152.638,E2 -1152.638} C_VEL
LIN {X 0,Y 594.61,Z 523.691,A -85,B 0,C 180,E1 -1153.829,E2 -1153.829} C_VEL
LIN {X 0,Y 595.022,Z 528.61,A -85,B 0,C 180,E1 -1153.907,E2 -1153.907} C_VEL
LIN {X 0,Y 594.863,Z 662.883,A -85,B 0,C 180,E1 -1155.569,E2 -1155.569} C_VEL
LIN {X 0,Y 594.804,Z 677.251,A -85,B 0,C 180,E1 -1155.891,E2 -1155.891} C_VEL
LIN {X 0,Y 594.735,Z 690.712,A -85,B 0,C 180,E1 -1156.329,E2 -1156.329} C_VEL
LIN {X 0,Y 594.654,Z 704.634,A -85,B 0,C 180,E1 -1156.936,E2 -1156.936} C_VEL
LIN {X 0,Y 594.581,Z 717.094,A -85,B 0,C 180,E1 -1157.629,E2 -1157.629} C_VEL
LIN {X 0,Y 594.524,Z 729.553,A -85,B 0,C 180,E1 -1158.487,E2 -1158.487} C_VEL
LIN {X 0,Y 594.449,Z 740.836,A -85,B 0,C 180,E1 -1159.441,E2 -1159.441} C_VEL
LIN {X 0,Y 594.368,Z 750.85,A -85,B 0,C 180,E1 -1160.471,E2 -1160.471} C_VEL
LIN {X 0,Y 594.324,Z 759.17,A -85,B 0,C 180,E1 -1161.5,E2 -1161.5} C_VEL
LIN {X 0,Y 594.303,Z 767.125,A -85,B 0,C 180,E1 -1162.696,E2 -1162.696} C_VEL
LIN {X 0,Y 594.279,Z 773.527,A -85,B 0,C 180,E1 -1163.89,E2 -1163.89} C_VEL
LIN {X 0,Y 594.237,Z 779.199,A -85,B 0,C 180,E1 -1165.251,E2 -1165.251} C_VEL
LIN {X 0,Y 594.259,Z 783.315,A -85,B 0,C 180,E1 -1166.61,E2 -1166.61} C_VEL
LIN {X 0,Y 594.238,Z 786,A -85,B 0,C 180,E1 -1167.967,E2 -1167.967} C_VEL
LIN {X 0,Y 594.237,Z 787.332,A -85,B 0,C 180,E1 -1169.322,E2 -1169.322} C_VEL
LIN {X 0,Y 594.237,Z 787.332,A -85,B 0,C 180,E1 -1170.678,E2 -1170.678} C_VEL
LIN {X 0,Y 594.238,Z 786,A -85,B 0,C 180,E1 -1172.033,E2 -1172.033} C_VEL
LIN {X 0,Y 594.259,Z 783.316,A -85,B 0,C 180,E1 -1173.39,E2 -1173.39} C_VEL
LIN {X 0,Y 594.237,Z 779.199,A -85,B 0,C 180,E1 -1174.749,E2 -1174.749} C_VEL
LIN {X 0,Y 594.279,Z 773.526,A -85,B 0,C 180,E1 -1176.11,E2 -1176.11} C_VEL
LIN {X 0,Y 594.303,Z 767.125,A -85,B 0,C 180,E1 -1177.304,E2 -1177.304} C_VEL
LIN {X 0,Y 594.324,Z 759.169,A -85,B 0,C 180,E1 -1178.5,E2 -1178.5} C_VEL
LIN {X 0,Y 594.367,Z 750.849,A -85,B 0,C 180,E1 -1179.529,E2 -1179.529} C_VEL
LIN {X 0,Y 594.449,Z 740.836,A -85,B 0,C 180,E1 -1180.559,E2 -1180.559} C_VEL
LIN {X 0,Y 594.524,Z 729.56,A -85,B 0,C 180,E1 -1181.512,E2 -1181.512} C_VEL
LIN {X 0,Y 594.562,Z 718.505,A -85,B 0,C 180,E1 -1182.285,E2 -1182.285} C_VEL
LIN {X 0,Y 594.651,Z 706.382,A -85,B 0,C 180,E1 -1182.977,E2 -1182.977} C_VEL
LIN {X 0,Y 594.747,Z 692.951,A -85,B 0,C 180,E1 -1183.583,E2 -1183.583} C_VEL
LIN {X 0,Y 594.798,Z 678.896,A -85,B 0,C 180,E1 -1184.062,E2 -1184.062} C_VEL
LIN {X 0,Y 594.85,Z 665.158,A -85,B 0,C 180,E1 -1184.388,E2 -1184.388} C_VEL
LIN {X 0,Y 594.893,Z 644.87,A -85,B 0,C 180,E1 -1184.671,E2 -1184.671} C_VEL
LIN {X 0,Y 594.926,Z 525.922,A -85,B 0,C 180,E1 -1186.129,E2 -1186.129} C_VEL
LIN {X 0,Y 594.61,Z 523.691,A -85,B 0,C 180,E1 -1186.171,E2 -1186.171} C_VEL
LIN {X 0,Y 594.745,Z 499.066,A -85,B 0,C 180,E1 -1188.9,E2 -1188.9} C_VEL
LIN {X 0,Y 594.887,Z 474.512,A -85,B 0,C 180,E1 -1191.666,E2 -1191.666} C_VEL
LIN {X 0,Y 594.758,Z 463.316,A -85,B 0,C 180,E1 -1192.951,E2 -1192.951} C_VEL
LIN {X 0,Y 594.401,Z 461.57,A -85,B 0,C 180,E1 -1193.196,E2 -1193.196} C_VEL
LIN {X 0,Y 594.392,Z 461.57,A -85,B 0,C 180,E1 -1196.024,E2 -1196.024} C_VEL
LIN {X 0,Y 594.385,Z 461.568,A -85,B 0,C 180,E1 -1198.958,E2 -1198.958} C_VEL
LIN {X 0,Y 594.395,Z 461.572,A -85,B 0,C 180,E1 -1201.645,E2 -1201.645} C_VEL
LIN {X 0,Y 594.379,Z 461.567,A -85,B 0,C 180,E1 -1204.58,E2 -1204.58} C_VEL
LIN {X 0,Y 594.393,Z 461.57,A -85,B 0,C 180,E1 -1207.609,E2 -1207.609} C_VEL
LIN {X 0,Y 594.37,Z 461.568,A -85,B 0,C 180,E1 -1210.567,E2 -1210.567} C_VEL
LIN {X 0,Y 594.383,Z 461.574,A -85,B 0,C 180,E1 -1213.298,E2 -1213.298} C_VEL
LIN {X 0,Y 594.363,Z 461.568,A -85,B 0,C 180,E1 -1216.161,E2 -1216.161} C_VEL
LIN {X 0,Y 594.382,Z 461.569,A -85,B 0,C 180,E1 -1218.536,E2 -1218.536} C_VEL
LIN {X 0,Y 594.391,Z 461.569,A -85,B 0,C 180,E1 -1221.295,E2 -1221.295} C_VEL
LIN {X 0,Y 594.356,Z 461.569,A -85,B 0,C 180,E1 -1223.756,E2 -1223.756} C_VEL
LIN {X 0,Y 594.382,Z 461.568,A -85,B 0,C 180,E1 -1226.239,E2 -1226.239} C_VEL
LIN {X 0,Y 594.395,Z 461.574,A -85,B 0,C 180,E1 -1228.651,E2 -1228.651} C_VEL
LIN {X 0,Y 594.388,Z 461.57,A -85,B 0,C 180,E1 -1231.042,E2 -1231.042} C_VEL
LIN {X 0,Y 594.392,Z 461.568,A -85,B 0,C 180,E1 -1233.977,E2 -1233.977} C_VEL
LIN {X 0,Y 594.389,Z 461.573,A -85,B 0,C 180,E1 -1236.296,E2 -1236.296} C_VEL
LIN {X 0,Y 594.393,Z 461.737,A -85,B 0,C 180,E1 -1237.222,E2 -1237.222} C_VEL
LIN {X 0,Y 594.846,Z 465.771,A -85,B 0,C 180,E1 -1237.786,E2 -1237.786} C_VEL
LIN {X 0,Y 594.697,Z 486.138,A -85,B 0,C 180,E1 -1240.497,E2 -1240.497} C_VEL
LIN {X 0,Y 594.617,Z 507.847,A -85,B 0,C 180,E1 -1243.339,E2 -1243.339} C_VEL
LIN {X 0,Y 594.518,Z 529.451,A -85,B 0,C 180,E1 -1246.124,E2 -1246.124} C_VEL
LIN {X 0,Y 594.433,Z 541.819,A -85,B 0,C 180,E1 -1247.702,E2 -1247.702} C_VEL
LIN {X 0,Y 594.773,Z 549.471,A -85,B 0,C 180,E1 -1247.806,E2 -1247.806} C_VEL
LIN {X 0,Y 594.651,Z 650.771,A -85,B 0,C 180,E1 -1249.049,E2 -1249.049} C_VEL
LIN {X 0,Y 594.654,Z 664.124,A -85,B 0,C 180,E1 -1249.358,E2 -1249.358} C_VEL
LIN {X 0,Y 594.547,Z 676.698,A -85,B 0,C 180,E1 -1249.787,E2 -1249.787} C_VEL
LIN {X 0,Y 594.541,Z 687.895,A -85,B 0,C 180,E1 -1250.302,E2 -1250.302} C_VEL
LIN {X 0,Y 594.452,Z 699.484,A -85,B 0,C 180,E1 -1250.987,E2 -1250.987} C_VEL
LIN {X 0,Y 594.421,Z 709.888,A -85,B 0,C 180,E1 -1251.758,E2 -1251.758} C_VEL
LIN {X 0,Y 594.379,Z 718.42,A -85,B 0,C 180,E1 -1252.527,E2 -1252.527} C_VEL
LIN {X 0,Y 594.345,Z 726.089,A -85,B 0,C 180,E1 -1253.358,E2 -1253.358} C_VEL
LIN {X 0,Y 594.31,Z 733.964,A -85,B 0,C 180,E1 -1254.401,E2 -1254.401} C_VEL
LIN {X 0,Y 594.277,Z 741.053,A -85,B 0,C 180,E1 -1255.591,E2 -1255.591} C_VEL
LIN {X 0,Y 594.271,Z 745.759,A -85,B 0,C 180,E1 -1256.61,E2 -1256.61} C_VEL
LIN {X 0,Y 594.256,Z 749.375,A -85,B 0,C 180,E1 -1257.628,E2 -1257.628} C_VEL
LIN {X 0,Y 594.248,Z 751.981,A -85,B 0,C 180,E1 -1258.645,E2 -1258.645} C_VEL
LIN {X 0,Y 594.239,Z 753.204,A -85,B 0,C 180,E1 -1259.322,E2 -1259.322} C_VEL
LIN {X 0,Y 594.237,Z 754.022,A -85,B 0,C 180,E1 -1260,E2 -1260} C_VEL
LIN {X 0,Y 594.248,Z 754.435,A -85,B 0,C 180,E1 -1261.355,E2 -1261.355} C_VEL
LIN {X 0,Y 594.239,Z 754.073,A -85,B 0,C 180,E1 -1262.033,E2 -1262.033} C_VEL
LIN {X 0,Y 594.222,Z 753.291,A -85,B 0,C 180,E1 -1262.712,E2 -1262.712} C_VEL
LIN {X 0,Y 594.26,Z 752.096,A -85,B 0,C 180,E1 -1263.39,E2 -1263.39} C_VEL
LIN {X 0,Y 594.265,Z 749.542,A -85,B 0,C 180,E1 -1264.409,E2 -1264.409} C_VEL
LIN {X 0,Y 594.277,Z 745.972,A -85,B 0,C 180,E1 -1265.429,E2 -1265.429} C_VEL
LIN {X 0,Y 594.263,Z 740.599,A -85,B 0,C 180,E1 -1266.584,E2 -1266.584} C_VEL
LIN {X 0,Y 594.298,Z 734.253,A -85,B 0,C 180,E1 -1267.645,E2 -1267.645} C_VEL
LIN {X 0,Y 594.356,Z 726.602,A -85,B 0,C 180,E1 -1268.671,E2 -1268.671} C_VEL
LIN {X 0,Y 594.354,Z 718.779,A -85,B 0,C 180,E1 -1269.529,E2 -1269.529} C_VEL
LIN {X 0,Y 594.425,Z 708.145,A -85,B 0,C 180,E1 -1270.474,E2 -1270.474} C_VEL
LIN {X 0,Y 594.471,Z 698.234,A -85,B 0,C 180,E1 -1271.185,E2 -1271.185} C_VEL
LIN {X 0,Y 594.543,Z 686.588,A -85,B 0,C 180,E1 -1271.852,E2 -1271.852} C_VEL
LIN {X 0,Y 594.596,Z 673.81,A -85,B 0,C 180,E1 -1272.414,E2 -1272.414} C_VEL
LIN {X 0,Y 594.604,Z 673.192,A -85,B 0,C 180,E1 -1272.437,E2 -1272.437} C_VEL
LIN {X 0,Y 593.999,Z 667.707,A -85,B 0,C 180,E1 -1272.643,E2 -1272.643} C_VEL
LIN {X 0,Y 591.201,Z 658.732,A -85,B 0,C 180,E1 -1272.952,E2 -1272.952} C_VEL
LIN {X 0,Y 588.39,Z 649.565,A -85,B 0,C 180,E1 -1273.192,E2 -1273.192} C_VEL
LIN {X 0,Y 587.759,Z 643.787,A -85,B 0,C 180,E1 -1273.287,E2 -1273.287} C_VEL
LIN {X 0,Y 587.786,Z 544.379,A -85,B 0,C 180,E1 -1274.507,E2 -1274.507} C_VEL
LIN {X 0,Y 587.413,Z 541.813,A -85,B 0,C 180,E1 -1274.552,E2 -1274.552} C_VEL
LIN {X 0,Y 587.6,Z 518.452,A -85,B 0,C 180,E1 -1277.578,E2 -1277.578} C_VEL
LIN {X 0,Y 587.709,Z 496.441,A -85,B 0,C 180,E1 -1280.474,E2 -1280.474} C_VEL
LIN {X 0,Y 587.888,Z 477.536,A -85,B 0,C 180,E1 -1282.999,E2 -1282.999} C_VEL
LIN {X 0,Y 587.821,Z 464.759,A -85,B 0,C 180,E1 -1284.737,E2 -1284.737} C_VEL
LIN {X 0,Y 587.341,Z 462.45,A -85,B 0,C 180,E1 -1285.09,E2 -1285.09} C_VEL
LIN {X 0,Y 587.343,Z 462.45,A -85,B 0,C 180,E1 -1287.818,E2 -1287.818} C_VEL
LIN {X 0,Y 587.338,Z 462.443,A -85,B 0,C 180,E1 -1290.509,E2 -1290.509} C_VEL
LIN {X 0,Y 587.336,Z 462.45,A -85,B 0,C 180,E1 -1293.397,E2 -1293.397} C_VEL
LIN {X 0,Y 587.297,Z 462.453,A -85,B 0,C 180,E1 -1295.9,E2 -1295.9} C_VEL
LIN {X 0,Y 587.326,Z 462.444,A -85,B 0,C 180,E1 -1298.48,E2 -1298.48} C_VEL
LIN {X 0,Y 587.336,Z 462.446,A -85,B 0,C 180,E1 -1301.157,E2 -1301.157} C_VEL
LIN {X 0,Y 587.314,Z 462.448,A -85,B 0,C 180,E1 -1304.112,E2 -1304.112} C_VEL
LIN {X 0,Y 587.326,Z 462.446,A -85,B 0,C 180,E1 -1306.994,E2 -1306.994} C_VEL
LIN {X 0,Y 587.315,Z 462.453,A -85,B 0,C 180,E1 -1309.745,E2 -1309.745} C_VEL
LIN {X 0,Y 587.348,Z 462.441,A -85,B 0,C 180,E1 -1312.392,E2 -1312.392} C_VEL
LIN {X 0,Y 587.362,Z 462.446,A -85,B 0,C 180,E1 -1315.78,E2 -1315.78} C_VEL
LIN {X 0,Y 587.345,Z 462.443,A -85,B 0,C 180,E1 -1318.231,E2 -1318.231} C_VEL
LIN {X 0,Y 587.352,Z 462.442,A -85,B 0,C 180,E1 -1320.866,E2 -1320.866} C_VEL
LIN {X 0,Y 587.36,Z 462.445,A -85,B 0,C 180,E1 -1323.819,E2 -1323.819} C_VEL
LIN {X 0,Y 587.333,Z 462.446,A -85,B 0,C 180,E1 -1325.993,E2 -1325.993} C_VEL
LIN {X 0,Y 587.325,Z 462.445,A -85,B 0,C 180,E1 -1328.226,E2 -1328.226} C_VEL
LIN {X 0,Y 587.354,Z 462.445,A -85,B 0,C 180,E1 -1331.151,E2 -1331.151} C_VEL
LIN {X 0,Y 587.329,Z 462.446,A -85,B 0,C 180,E1 -1334.025,E2 -1334.025} C_VEL
LIN {X 0,Y 587.362,Z 462.441,A -85,B 0,C 180,E1 -1336.154,E2 -1336.154} C_VEL
LIN {X 0,Y 587.348,Z 462.444,A -85,B 0,C 180,E1 -1338.962,E2 -1338.962} C_VEL
LIN {X 0,Y 587.373,Z 462.444,A -85,B 0,C 180,E1 -1341.745,E2 -1341.745} C_VEL
LIN {X 0,Y 587.356,Z 462.44,A -85,B 0,C 180,E1 -1344.507,E2 -1344.507} C_VEL
LIN {X 0,Y 587.381,Z 462.444,A -85,B 0,C 180,E1 -1347.257,E2 -1347.257} C_VEL
LIN {X 0,Y 587.386,Z 462.439,A -85,B 0,C 180,E1 -1350,E2 -1350} C_VEL
LIN {X 0,Y 587.372,Z 462.439,A -85,B 0,C 180,E1 -1352.743,E2 -1352.743} C_VEL
LIN {X 0,Y 587.369,Z 462.448,A -85,B 0,C 180,E1 -1355.493,E2 -1355.493} C_VEL
LIN {X 0,Y 587.367,Z 462.439,A -85,B 0,C 180,E1 -1358.255,E2 -1358.255} C_VEL
LIN {X 0,Y 587.351,Z 462.447,A -85,B 0,C 180,E1 -1361.134,E2 -1361.134} C_VEL
LIN {X 0,Y 587.368,Z 462.439,A -85,B 0,C 180,E1 -1364.261,E2 -1364.261} C_VEL
LIN {X 0,Y 587.351,Z 462.452,A -85,B 0,C 180,E1 -1367.406,E2 -1367.406} C_VEL
LIN {X 0,Y 587.33,Z 462.443,A -85,B 0,C 180,E1 -1370.305,E2 -1370.305} C_VEL
LIN {X 0,Y 587.325,Z 462.453,A -85,B 0,C 180,E1 -1373.259,E2 -1373.259} C_VEL
LIN {X 0,Y 587.336,Z 462.451,A -85,B 0,C 180,E1 -1375.517,E2 -1375.517} C_VEL
LIN {X 0,Y 587.348,Z 462.444,A -85,B 0,C 180,E1 -1377.818,E2 -1377.818} C_VEL
LIN {X 0,Y 587.342,Z 462.442,A -85,B 0,C 180,E1 -1380.51,E2 -1380.51} C_VEL
LIN {X 0,Y 587.337,Z 462.452,A -85,B 0,C 180,E1 -1383.397,E2 -1383.397} C_VEL
LIN {X 0,Y 587.293,Z 462.45,A -85,B 0,C 180,E1 -1385.9,E2 -1385.9} C_VEL
LIN {X 0,Y 587.334,Z 462.443,A -85,B 0,C 180,E1 -1388.479,E2 -1388.479} C_VEL
LIN {X 0,Y 587.339,Z 462.45,A -85,B 0,C 180,E1 -1391.157,E2 -1391.157} C_VEL
LIN {X 0,Y 587.337,Z 462.443,A -85,B 0,C 180,E1 -1394.114,E2 -1394.114} C_VEL
LIN {X 0,Y 587.314,Z 462.451,A -85,B 0,C 180,E1 -1396.993,E2 -1396.993} C_VEL
LIN {X 0,Y 587.318,Z 462.448,A -85,B 0,C 180,E1 -1399.746,E2 -1399.746} C_VEL
LIN {X 0,Y 587.345,Z 462.442,A -85,B 0,C 180,E1 -1402.392,E2 -1402.392} C_VEL
LIN {X 0,Y 587.369,Z 462.441,A -85,B 0,C 180,E1 -1405.78,E2 -1405.78} C_VEL
LIN {X 0,Y 587.342,Z 462.442,A -85,B 0,C 180,E1 -1408.231,E2 -1408.231} C_VEL
LIN {X 0,Y 587.353,Z 462.445,A -85,B 0,C 180,E1 -1410.867,E2 -1410.867} C_VEL
LIN {X 0,Y 587.364,Z 462.443,A -85,B 0,C 180,E1 -1413.819,E2 -1413.819} C_VEL
LIN {X 0,Y 587.383,Z 462.589,A -85,B 0,C 180,E1 -1415.809,E2 -1415.809} C_VEL
LIN {X 0,Y 587.982,Z 466.743,A -85,B 0,C 180,E1 -1416.396,E2 -1416.396} C_VEL
LIN {X 0,Y 587.848,Z 488.951,A -85,B 0,C 180,E1 -1419.348,E2 -1419.348} C_VEL
LIN {X 0,Y 587.631,Z 512.549,A -85,B 0,C 180,E1 -1422.423,E2 -1422.423} C_VEL
LIN {X 0,Y 587.511,Z 534.76,A -85,B 0,C 180,E1 -1425.274,E2 -1425.274} C_VEL
LIN {X 0,Y 587.437,Z 544.737,A -85,B 0,C 180,E1 -1426.542,E2 -1426.542} C_VEL
LIN {X 0,Y 587.892,Z 550.927,A -85,B 0,C 180,E1 -1426.63,E2 -1426.63} C_VEL
LIN {X 0,Y 587.739,Z 653.264,A -85,B 0,C 180,E1 -1427.899,E2 -1427.899} C_VEL
LIN {X 0,Y 587.663,Z 666.706,A -85,B 0,C 180,E1 -1428.204,E2 -1428.204} C_VEL
LIN {X 0,Y 587.595,Z 679.544,A -85,B 0,C 180,E1 -1428.646,E2 -1428.646} C_VEL
LIN {X 0,Y 587.532,Z 691.898,A -85,B 0,C 180,E1 -1429.228,E2 -1429.228} C_VEL
LIN {X 0,Y 587.455,Z 703.327,A -85,B 0,C 180,E1 -1429.923,E2 -1429.923} C_VEL
LIN {X 0,Y 587.385,Z 713.6,A -85,B 0,C 180,E1 -1430.705,E2 -1430.705} C_VEL
LIN {X 0,Y 587.341,Z 722.844,A -85,B 0,C 180,E1 -1431.571,E2 -1431.571} C_VEL
LIN {X 0,Y 587.259,Z 731.837,A -85,B 0,C 180,E1 -1432.608,E2 -1432.608} C_VEL
LIN {X 0,Y 587.199,Z 738.945,A -85,B 0,C 180,E1 -1433.624,E2 -1433.624} C_VEL
LIN {X 0,Y 587.211,Z 743.95,A -85,B 0,C 180,E1 -1434.506,E2 -1434.506} C_VEL
LIN {X 0,Y 587.188,Z 748.693,A -85,B 0,C 180,E1 -1435.538,E2 -1435.538} C_VEL
LIN {X 0,Y 587.194,Z 752.324,A -85,B 0,C 180,E1 -1436.569,E2 -1436.569} C_VEL
LIN {X 0,Y 587.131,Z 754.186,A -85,B 0,C 180,E1 -1437.256,E2 -1437.256} C_VEL
LIN {X 0,Y 587.139,Z 755.611,A -85,B 0,C 180,E1 -1437.942,E2 -1437.942} C_VEL
LIN {X 0,Y 587.147,Z 756.636,A -85,B 0,C 180,E1 -1438.628,E2 -1438.628} C_VEL
LIN {X 0,Y 587.14,Z 757.253,A -85,B 0,C 180,E1 -1439.314,E2 -1439.314} C_VEL
LIN {X 0,Y 587.14,Z 757.313,A -85,B 0,C 180,E1 -1440.686,E2 -1440.686} C_VEL
LIN {X 0,Y 587.147,Z 756.738,A -85,B 0,C 180,E1 -1441.372,E2 -1441.372} C_VEL
LIN {X 0,Y 587.133,Z 754.413,A -85,B 0,C 180,E1 -1442.744,E2 -1442.744} C_VEL
LIN {X 0,Y 587.213,Z 751.542,A -85,B 0,C 180,E1 -1443.774,E2 -1443.774} C_VEL
LIN {X 0,Y 587.147,Z 747.642,A -85,B 0,C 180,E1 -1444.806,E2 -1444.806} C_VEL
LIN {X 0,Y 587.229,Z 742.603,A -85,B 0,C 180,E1 -1445.839,E2 -1445.839} C_VEL
LIN {X 0,Y 587.229,Z 736.253,A -85,B 0,C 180,E1 -1446.874,E2 -1446.874} C_VEL
LIN {X 0,Y 587.288,Z 728.368,A -85,B 0,C 180,E1 -1447.91,E2 -1447.91} C_VEL
LIN {X 0,Y 587.343,Z 718.52,A -85,B 0,C 180,E1 -1448.949,E2 -1448.949} C_VEL
LIN {X 0,Y 587.409,Z 708.169,A -85,B 0,C 180,E1 -1449.816,E2 -1449.816} C_VEL
LIN {X 0,Y 587.498,Z 697.967,A -85,B 0,C 180,E1 -1450.511,E2 -1450.511} C_VEL
LIN {X 0,Y 587.577,Z 686.993,A -85,B 0,C 180,E1 -1451.112,E2 -1451.112} C_VEL
LIN {X 0,Y 587.634,Z 674.368,A -85,B 0,C 180,E1 -1451.64,E2 -1451.64} C_VEL
LIN {X 0,Y 587.718,Z 661.775,A -85,B 0,C 180,E1 -1452.014,E2 -1452.014} C_VEL
LIN {X 0,Y 587.773,Z 649.18,A -85,B 0,C 180,E1 -1452.253,E2 -1452.253} C_VEL
LIN {X 0,Y 587.755,Z 546.836,A -85,B 0,C 180,E1 -1453.514,E2 -1453.514} C_VEL
LIN {X 0,Y 587.422,Z 544.665,A -85,B 0,C 180,E1 -1453.558,E2 -1453.558} C_VEL
LIN {X 0,Y 587.568,Z 524.354,A -85,B 0,C 180,E1 -1456.147,E2 -1456.147} C_VEL
LIN {X 0,Y 587.708,Z 502.136,A -85,B 0,C 180,E1 -1459.018,E2 -1459.018} C_VEL
LIN {X 0,Y 587.886,Z 479.912,A -85,B 0,C 180,E1 -1461.937,E2 -1461.937} C_VEL
LIN {X 0,Y 588.019,Z 466.022,A -85,B 0,C 180,E1 -1463.79,E2 -1463.79} C_VEL
LIN {X 0,Y 587.364,Z 462.448,A -85,B 0,C 180,E1 -1464.316,E2 -1464.316} C_VEL
LIN {X 0,Y 587.331,Z 462.451,A -85,B 0,C 180,E1 -1467.046,E2 -1467.046} C_VEL
LIN {X 0,Y 587.35,Z 462.444,A -85,B 0,C 180,E1 -1469.379,E2 -1469.379} C_VEL
LIN {X 0,Y 587.345,Z 462.443,A -85,B 0,C 180,E1 -1471.835,E2 -1471.835} C_VEL
LIN {X 0,Y 587.352,Z 462.447,A -85,B 0,C 180,E1 -1474.348,E2 -1474.348} C_VEL
LIN {X 0,Y 587.345,Z 462.442,A -85,B 0,C 180,E1 -1477.608,E2 -1477.608} C_VEL
LIN {X 0,Y 587.318,Z 462.45,A -85,B 0,C 180,E1 -1480.254,E2 -1480.254} C_VEL
LIN {X 0,Y 587.315,Z 462.448,A -85,B 0,C 180,E1 -1483.118,E2 -1483.118} C_VEL
LIN {X 0,Y 587.338,Z 462.446,A -85,B 0,C 180,E1 -1486.051,E2 -1486.051} C_VEL
LIN {X 0,Y 587.339,Z 462.446,A -85,B 0,C 180,E1 -1488.925,E2 -1488.925} C_VEL
LIN {X 0,Y 587.332,Z 462.444,A -85,B 0,C 180,E1 -1491.521,E2 -1491.521} C_VEL
LIN {X 0,Y 587.35,Z 462.447,A -85,B 0,C 180,E1 -1494.104,E2 -1494.104} C_VEL
LIN {X 0,Y 587.342,Z 462.445,A -85,B 0,C 180,E1 -1496.888,E2 -1496.888} C_VEL
LIN {X 0,Y 587.354,Z 462.442,A -85,B 0,C 180,E1 -1499.488,E2 -1499.488} C_VEL
LIN {X 0,Y 587.354,Z 462.451,A -85,B 0,C 180,E1 -1502.307,E2 -1502.307} C_VEL
LIN {X 0,Y 587.34,Z 462.451,A -85,B 0,C 180,E1 -1504.484,E2 -1504.484} C_VEL
LIN {X 0,Y 587.377,Z 462.518,A -85,B 0,C 180,E1 -1506.65,E2 -1506.65} C_VEL
LIN {X 0,Y 588.081,Z 467.49,A -85,B 0,C 180,E1 -1507.258,E2 -1507.258} C_VEL
LIN {X 0,Y 587.874,Z 490.506,A -85,B 0,C 180,E1 -1509.897,E2 -1509.897} C_VEL
LIN {X 0,Y 587.699,Z 515.856,A -85,B 0,C 180,E1 -1512.757,E2 -1512.757} C_VEL
LIN {X 0,Y 587.643,Z 523.691,A -85,B 0,C 180,E1 -1513.632,E2 -1513.632} C_VEL
LIN {X 0,Y 588.21,Z 528.61,A -85,B 0,C 180,E1 -1513.715,E2 -1513.715} C_VEL
LIN {X 0,Y 587.994,Z 662.883,A -85,B 0,C 180,E1 -1515.397,E2 -1515.397} C_VEL
LIN {X 0,Y 587.913,Z 677.44,A -85,B 0,C 180,E1 -1515.728,E2 -1515.728} C_VEL
LIN {X 0,Y 587.824,Z 691.835,A -85,B 0,C 180,E1 -1516.209,E2 -1516.209} C_VEL
LIN {X 0,Y 587.731,Z 704.636,A -85,B 0,C 180,E1 -1516.78,E2 -1516.78} C_VEL
LIN {X 0,Y 587.605,Z 717.096,A -85,B 0,C 180,E1 -1517.48,E2 -1517.48} C_VEL
LIN {X 0,Y 587.513,Z 728.475,A -85,B 0,C 180,E1 -1518.267,E2 -1518.267} C_VEL
LIN {X 0,Y 587.467,Z 738.933,A -85,B 0,C 180,E1 -1519.139,E2 -1519.139} C_VEL
LIN {X 0,Y 587.353,Z 749.334,A -85,B 0,C 180,E1 -1520.183,E2 -1520.183} C_VEL
LIN {X 0,Y 587.311,Z 757.913,A -85,B 0,C 180,E1 -1521.224,E2 -1521.224} C_VEL
LIN {X 0,Y 587.249,Z 766.115,A -85,B 0,C 180,E1 -1522.435,E2 -1522.435} C_VEL
LIN {X 0,Y 587.179,Z 772.681,A -85,B 0,C 180,E1 -1523.635,E2 -1523.635} C_VEL
LIN {X 0,Y 587.16,Z 777.961,A -85,B 0,C 180,E1 -1524.85,E2 -1524.85} C_VEL
LIN {X 0,Y 587.179,Z 781.442,A -85,B 0,C 180,E1 -1525.882,E2 -1525.882} C_VEL
LIN {X 0,Y 587.13,Z 784.831,A -85,B 0,C 180,E1 -1527.256,E2 -1527.256} C_VEL
LIN {X 0,Y 587.141,Z 786.832,A -85,B 0,C 180,E1 -1528.628,E2 -1528.628} C_VEL
LIN {X 0,Y 587.135,Z 787.5,A -85,B 0,C 180,E1 -1530,E2 -1530} C_VEL
LIN {X 0,Y 587.141,Z 786.832,A -85,B 0,C 180,E1 -1531.372,E2 -1531.372} C_VEL
LIN {X 0,Y 587.13,Z 784.832,A -85,B 0,C 180,E1 -1532.744,E2 -1532.744} C_VEL
LIN {X 0,Y 587.179,Z 781.443,A -85,B 0,C 180,E1 -1534.118,E2 -1534.118} C_VEL
LIN {X 0,Y 587.199,Z 776.567,A -85,B 0,C 180,E1 -1535.495,E2 -1535.495} C_VEL
LIN {X 0,Y 587.209,Z 770.051,A -85,B 0,C 180,E1 -1536.874,E2 -1536.874} C_VEL
LIN {X 0,Y 587.269,Z 762.799,A -85,B 0,C 180,E1 -1538.084,E2 -1538.084} C_VEL
LIN {X 0,Y 587.322,Z 753.822,A -85,B 0,C 180,E1 -1539.297,E2 -1539.297} C_VEL
LIN {X 0,Y 587.372,Z 744.39,A -85,B 0,C 180,E1 -1540.339,E2 -1540.339} C_VEL
LIN {X 0,Y 587.475,Z 734.025,A -85,B 0,C 180,E1 -1541.29,E2 -1541.29} C_VEL
LIN {X 0,Y 587.575,Z 722.428,A -85,B 0,C 180,E1 -1542.17,E2 -1542.17} C_VEL
LIN {X 0,Y 587.67,Z 709.646,A -85,B 0,C 180,E1 -1542.958,E2 -1542.958} C_VEL
LIN {X 0,Y 587.814,Z 697.158,A -85,B 0,C 180,E1 -1543.57,E2 -1543.57} C_VEL
LIN {X 0,Y 587.902,Z 683.725,A -85,B 0,C 180,E1 -1544.081,E2 -1544.081} C_VEL
LIN {X 0,Y 587.963,Z 669.297,A -85,B 0,C 180,E1 -1544.477,E2 -1544.477} C_VEL
LIN {X 0,Y 588.013,Z 655.591,A -85,B 0,C 180,E1 -1544.713,E2 -1544.713} C_VEL
LIN {X 0,Y 588.129,Z 526.815,A -85,B 0,C 180,E1 -1546.309,E2 -1546.309} C_VEL
LIN {X 0,Y 587.654,Z 523.691,A -85,B 0,C 180,E1 -1546.367,E2 -1546.367} C_VEL
LIN {X 0,Y 587.818,Z 498.701,A -85,B 0,C 180,E1 -1549.173,E2 -1549.173} C_VEL
LIN {X 0,Y 588.031,Z 474.512,A -85,B 0,C 180,E1 -1551.931,E2 -1551.931} C_VEL
LIN {X 0,Y 587.942,Z 465.216,A -85,B 0,C 180,E1 -1553.012,E2 -1553.012} C_VEL
LIN {X 0,Y 587.36,Z 462.449,A -85,B 0,C 180,E1 -1553.374,E2 -1553.374} C_VEL
LIN {X 0,Y 587.344,Z 462.445,A -85,B 0,C 180,E1 -1556.279,E2 -1556.279} C_VEL
LIN {X 0,Y 587.352,Z 462.446,A -85,B 0,C 180,E1 -1559.134,E2 -1559.134} C_VEL
LIN {X 0,Y 587.357,Z 462.446,A -85,B 0,C 180,E1 -1561.837,E2 -1561.837} C_VEL
LIN {X 0,Y 587.348,Z 462.443,A -85,B 0,C 180,E1 -1564.348,E2 -1564.348} C_VEL
LIN {X 0,Y 587.348,Z 462.448,A -85,B 0,C 180,E1 -1567.608,E2 -1567.608} C_VEL
LIN {X 0,Y 587.314,Z 462.447,A -85,B 0,C 180,E1 -1570.255,E2 -1570.255} C_VEL
LIN {X 0,Y 587.328,Z 462.454,A -85,B 0,C 180,E1 -1573.119,E2 -1573.119} C_VEL
LIN {X 0,Y 587.315,Z 462.446,A -85,B 0,C 180,E1 -1576.049,E2 -1576.049} C_VEL
LIN {X 0,Y 587.339,Z 462.452,A -85,B 0,C 180,E1 -1578.925,E2 -1578.925} C_VEL
LIN {X 0,Y 587.335,Z 462.446,A -85,B 0,C 180,E1 -1581.521,E2 -1581.521} C_VEL
LIN {X 0,Y 587.298,Z 462.449,A -85,B 0,C 180,E1 -1584.1,E2 -1584.1} C_VEL
LIN {X 0,Y 587.339,Z 462.451,A -85,B 0,C 180,E1 -1586.604,E2 -1586.604} C_VEL
LIN {X 0,Y 587.345,Z 462.448,A -85,B 0,C 180,E1 -1589.034,E2 -1589.034} C_VEL
LIN {X 0,Y 587.327,Z 462.447,A -85,B 0,C 180,E1 -1591.403,E2 -1591.403} C_VEL
LIN {X 0,Y 587.365,Z 462.443,A -85,B 0,C 180,E1 -1593.819,E2 -1593.819} C_VEL
LIN {X 0,Y 587.338,Z 462.448,A -85,B 0,C 180,E1 -1595.994,E2 -1595.994} C_VEL
LIN {X 0,Y 587.365,Z 462.579,A -85,B 0,C 180,E1 -1597.034,E2 -1597.034} C_VEL
LIN {X 0,Y 587.973,Z 467.233,A -85,B 0,C 180,E1 -1597.697,E2 -1597.697} C_VEL
LIN {X 0,Y 587.771,Z 487.601,A -85,B 0,C 180,E1 -1600.44,E2 -1600.44} C_VEL
LIN {X 0,Y 587.647,Z 509.347,A -85,B 0,C 180,E1 -1603.32,E2 -1603.32} C_VEL
LIN {X 0,Y 587.527,Z 531.114,A -85,B 0,C 180,E1 -1606.158,E2 -1606.158} C_VEL
LIN {X 0,Y 587.43,Z 541.836,A -85,B 0,C 180,E1 -1607.542,E2 -1607.542} C_VEL
LIN {X 0,Y 587.876,Z 548.738,A -85,B 0,C 180,E1 -1607.639,E2 -1607.639} C_VEL
LIN {X 0,Y 587.719,Z 651.106,A -85,B 0,C 180,E1 -1608.912,E2 -1608.912} C_VEL
LIN {X 0,Y 587.711,Z 664.567,A -85,B 0,C 180,E1 -1609.231,E2 -1609.231} C_VEL
LIN {X 0,Y 587.568,Z 676.996,A -85,B 0,C 180,E1 -1609.664,E2 -1609.664} C_VEL
LIN {X 0,Y 587.556,Z 688.138,A -85,B 0,C 180,E1 -1610.186,E2 -1610.186} C_VEL
LIN {X 0,Y 587.45,Z 699.675,A -85,B 0,C 180,E1 -1610.879,E2 -1610.879} C_VEL
LIN {X 0,Y 587.405,Z 710.044,A -85,B 0,C 180,E1 -1611.659,E2 -1611.659} C_VEL
LIN {X 0,Y 587.32,Z 718.553,A -85,B 0,C 180,E1 -1612.436,E2 -1612.436} C_VEL
LIN {X 0,Y 587.271,Z 726.848,A -85,B 0,C 180,E1 -1613.356,E2 -1613.356} C_VEL
LIN {X 0,Y 587.239,Z 734.045,A -85,B 0,C 180,E1 -1614.334,E2 -1614.334} C_VEL
LIN {X 0,Y 587.2,Z 741.122,A -85,B 0,C 180,E1 -1615.538,E2 -1615.538} C_VEL
LIN {X 0,Y 587.197,Z 745.811,A -85,B 0,C 180,E1 -1616.569,E2 -1616.569} C_VEL
LIN {X 0,Y 587.173,Z 749.417,A -85,B 0,C 180,E1 -1617.599,E2 -1617.599} C_VEL
LIN {X 0,Y 587.148,Z 752.007,A -85,B 0,C 180,E1 -1618.628,E2 -1618.628} C_VEL
LIN {X 0,Y 587.14,Z 753.221,A -85,B 0,C 180,E1 -1619.314,E2 -1619.314} C_VEL
LIN {X 0,Y 587.138,Z 754.03,A -85,B 0,C 180,E1 -1620,E2 -1620} C_VEL
LIN {X 0,Y 587.147,Z 754.432,A -85,B 0,C 180,E1 -1621.372,E2 -1621.372} C_VEL
LIN {X 0,Y 587.138,Z 754.059,A -85,B 0,C 180,E1 -1622.058,E2 -1622.058} C_VEL
LIN {X 0,Y 587.128,Z 753.269,A -85,B 0,C 180,E1 -1622.744,E2 -1622.744} C_VEL
LIN {X 0,Y 587.183,Z 752.07,A -85,B 0,C 180,E1 -1623.431,E2 -1623.431} C_VEL
LIN {X 0,Y 587.183,Z 749.505,A -85,B 0,C 180,E1 -1624.462,E2 -1624.462} C_VEL
LIN {X 0,Y 587.201,Z 745.918,A -85,B 0,C 180,E1 -1625.494,E2 -1625.494} C_VEL
LIN {X 0,Y 587.179,Z 740.921,A -85,B 0,C 180,E1 -1626.59,E2 -1626.59} C_VEL
LIN {X 0,Y 587.234,Z 734.169,A -85,B 0,C 180,E1 -1627.738,E2 -1627.738} C_VEL
LIN {X 0,Y 587.287,Z 726.492,A -85,B 0,C 180,E1 -1628.776,E2 -1628.776} C_VEL
LIN {X 0,Y 587.353,Z 716.868,A -85,B 0,C 180,E1 -1629.817,E2 -1629.817} C_VEL
LIN {X 0,Y 587.423,Z 706.9,A -85,B 0,C 180,E1 -1630.687,E2 -1630.687} C_VEL
LIN {X 0,Y 587.484,Z 695.649,A -85,B 0,C 180,E1 -1631.471,E2 -1631.471} C_VEL
LIN {X 0,Y 587.584,Z 684.571,A -85,B 0,C 180,E1 -1632.082,E2 -1632.082} C_VEL
LIN {X 0,Y 587.651,Z 672.302,A -85,B 0,C 180,E1 -1632.607,E2 -1632.607} C_VEL
LIN {X 0,Y 587.688,Z 659.389,A -85,B 0,C 180,E1 -1633.001,E2 -1633.001} C_VEL
LIN {X 0,Y 587.728,Z 647.019,A -85,B 0,C 180,E1 -1633.242,E2 -1633.242} C_VEL
LIN {X 0,Y 587.759,Z 643.787,A -85,B 0,C 180,E1 -1633.287,E2 -1633.287} C_VEL
LIN {X 0,Y 587.137,Z 637.977,A -85,B 0,C 180,E1 -1633.371,E2 -1633.371} C_VEL
LIN {X 0,Y 581.526,Z 619.284,A -85,B 0,C 180,E1 -1633.724,E2 -1633.724} C_VEL
LIN {X 0,Y 580.86,Z 613.475,A -85,B 0,C 180,E1 -1633.811,E2 -1633.811} C_VEL
LIN {X 0,Y 580.829,Z 544.575,A -85,B 0,C 180,E1 -1634.668,E2 -1634.668} C_VEL
LIN {X 0,Y 580.397,Z 541.71,A -85,B 0,C 180,E1 -1634.731,E2 -1634.731} C_VEL
LIN {X 0,Y 580.617,Z 519.723,A -85,B 0,C 180,E1 -1637.614,E2 -1637.614} C_VEL
LIN {X 0,Y 580.784,Z 497.713,A -85,B 0,C 180,E1 -1640.544,E2 -1640.544} C_VEL
LIN {X 0,Y 581.002,Z 477.415,A -85,B 0,C 180,E1 -1643.289,E2 -1643.289} C_VEL
LIN {X 0,Y 581.08,Z 468.016,A -85,B 0,C 180,E1 -1644.579,E2 -1644.579} C_VEL
LIN {X 0,Y 580.324,Z 463.322,A -85,B 0,C 180,E1 -1645.271,E2 -1645.271} C_VEL
LIN {X 0,Y 580.299,Z 463.323,A -85,B 0,C 180,E1 -1648.186,E2 -1648.186} C_VEL
LIN {X 0,Y 580.286,Z 463.322,A -85,B 0,C 180,E1 -1650.694,E2 -1650.694} C_VEL
LIN {X 0,Y 580.306,Z 463.325,A -85,B 0,C 180,E1 -1653.316,E2 -1653.316} C_VEL
LIN {X 0,Y 580.263,Z 463.332,A -85,B 0,C 180,E1 -1655.758,E2 -1655.758} C_VEL
LIN {X 0,Y 580.288,Z 463.323,A -85,B 0,C 180,E1 -1658.146,E2 -1658.146} C_VEL
LIN {X 0,Y 580.3,Z 463.32,A -85,B 0,C 180,E1 -1660.843,E2 -1660.843} C_VEL
LIN {X 0,Y 580.275,Z 463.332,A -85,B 0,C 180,E1 -1663.658,E2 -1663.658} C_VEL
LIN {X 0,Y 580.289,Z 463.32,A -85,B 0,C 180,E1 -1666.608,E2 -1666.608} C_VEL
LIN {X 0,Y 580.3,Z 463.323,A -85,B 0,C 180,E1 -1669.156,E2 -1669.156} C_VEL
LIN {X 0,Y 580.293,Z 463.324,A -85,B 0,C 180,E1 -1671.927,E2 -1671.927} C_VEL
LIN {X 0,Y 580.252,Z 463.325,A -85,B 0,C 180,E1 -1674.452,E2 -1674.452} C_VEL
LIN {X 0,Y 580.293,Z 463.322,A -85,B 0,C 180,E1 -1676.975,E2 -1676.975} C_VEL
LIN {X 0,Y 580.298,Z 463.328,A -85,B 0,C 180,E1 -1679.425,E2 -1679.425} C_VEL
LIN {X 0,Y 580.301,Z 463.321,A -85,B 0,C 180,E1 -1682.141,E2 -1682.141} C_VEL
LIN {X 0,Y 580.324,Z 463.322,A -85,B 0,C 180,E1 -1685.27,E2 -1685.27} C_VEL
LIN {X 0,Y 580.275,Z 463.326,A -85,B 0,C 180,E1 -1687.947,E2 -1687.947} C_VEL
LIN {X 0,Y 580.322,Z 463.318,A -85,B 0,C 180,E1 -1690.914,E2 -1690.914} C_VEL
LIN {X 0,Y 580.283,Z 463.326,A -85,B 0,C 180,E1 -1693.826,E2 -1693.826} C_VEL
LIN {X 0,Y 580.329,Z 463.318,A -85,B 0,C 180,E1 -1695.983,E2 -1695.983} C_VEL
LIN {X 0,Y 580.307,Z 463.32,A -85,B 0,C 180,E1 -1698.827,E2 -1698.827} C_VEL
LIN {X 0,Y 580.337,Z 463.322,A -85,B 0,C 180,E1 -1701.644,E2 -1701.644} C_VEL
LIN {X 0,Y 580.323,Z 463.316,A -85,B 0,C 180,E1 -1704.44,E2 -1704.44} C_VEL
LIN {X 0,Y 580.347,Z 463.32,A -85,B 0,C 180,E1 -1707.223,E2 -1707.223} C_VEL
LIN {X 0,Y 580.355,Z 463.314,A -85,B 0,C 180,E1 -1710,E2 -1710} C_VEL
LIN {X 0,Y 580.339,Z 463.316,A -85,B 0,C 180,E1 -1712.777,E2 -1712.777} C_VEL
LIN {X 0,Y 580.335,Z 463.323,A -85,B 0,C 180,E1 -1715.56,E2 -1715.56} C_VEL
LIN {X 0,Y 580.33,Z 463.315,A -85,B 0,C 180,E1 -1718.356,E2 -1718.356} C_VEL
LIN {X 0,Y 580.302,Z 463.325,A -85,B 0,C 180,E1 -1721.191,E2 -1721.191} C_VEL
LIN {X 0,Y 580.33,Z 463.317,A -85,B 0,C 180,E1 -1724.017,E2 -1724.017} C_VEL
LIN {X 0,Y 580.315,Z 463.32,A -85,B 0,C 180,E1 -1726.914,E2 -1726.914} C_VEL
LIN {X 0,Y 580.307,Z 463.322,A -85,B 0,C 180,E1 -1729.822,E2 -1729.822} C_VEL
LIN {X 0,Y 580.297,Z 463.321,A -85,B 0,C 180,E1 -1732.802,E2 -1732.802} C_VEL
LIN {X 0,Y 580.309,Z 463.324,A -85,B 0,C 180,E1 -1735.08,E2 -1735.08} C_VEL
LIN {X 0,Y 580.3,Z 463.319,A -85,B 0,C 180,E1 -1738.186,E2 -1738.186} C_VEL
LIN {X 0,Y 580.291,Z 463.322,A -85,B 0,C 180,E1 -1740.695,E2 -1740.695} C_VEL
LIN {X 0,Y 580.306,Z 463.329,A -85,B 0,C 180,E1 -1743.317,E2 -1743.317} C_VEL
LIN {X 0,Y 580.248,Z 463.329,A -85,B 0,C 180,E1 -1745.756,E2 -1745.756} C_VEL
LIN {X 0,Y 580.291,Z 463.321,A -85,B 0,C 180,E1 -1748.146,E2 -1748.146} C_VEL
LIN {X 0,Y 580.302,Z 463.322,A -85,B 0,C 180,E1 -1750.843,E2 -1750.843} C_VEL
LIN {X 0,Y 580.291,Z 463.325,A -85,B 0,C 180,E1 -1753.657,E2 -1753.657} C_VEL
LIN {X 0,Y 580.275,Z 463.323,A -85,B 0,C 180,E1 -1756.61,E2 -1756.61} C_VEL
LIN {X 0,Y 580.3,Z 463.327,A -85,B 0,C 180,E1 -1759.157,E2 -1759.157} C_VEL
LIN {X 0,Y 580.291,Z 463.322,A -85,B 0,C 180,E1 -1761.927,E2 -1761.927} C_VEL
LIN {X 0,Y 580.26,Z 463.324,A -85,B 0,C 180,E1 -1764.453,E2 -1764.453} C_VEL
LIN {X 0,Y 580.292,Z 463.326,A -85,B 0,C 180,E1 -1766.975,E2 -1766.975} C_VEL
LIN {X 0,Y 580.297,Z 463.327,A -85,B 0,C 180,E1 -1769.425,E2 -1769.425} C_VEL
LIN {X 0,Y 580.295,Z 463.32,A -85,B 0,C 180,E1 -1772.143,E2 -1772.143} C_VEL
LIN {X 0,Y 580.31,Z 463.325,A -85,B 0,C 180,E1 -1774.92,E2 -1774.92} C_VEL
LIN {X 0,Y 580.375,Z 463.512,A -85,B 0,C 180,E1 -1775.624,E2 -1775.624} C_VEL
LIN {X 0,Y 581.124,Z 468.135,A -85,B 0,C 180,E1 -1776.289,E2 -1776.289} C_VEL
LIN {X 0,Y 580.911,Z 488.956,A -85,B 0,C 180,E1 -1779.09,E2 -1779.09} C_VEL
LIN {X 0,Y 580.726,Z 509.777,A -85,B 0,C 180,E1 -1781.843,E2 -1781.843} C_VEL
LIN {X 0,Y 580.515,Z 531.988,A -85,B 0,C 180,E1 -1784.733,E2 -1784.733} C_VEL
LIN {X 0,Y 580.429,Z 544.742,A -85,B 0,C 180,E1 -1786.376,E2 -1786.376} C_VEL
LIN {X 0,Y 580.999,Z 550.973,A -85,B 0,C 180,E1 -1786.468,E2 -1786.468} C_VEL
LIN {X 0,Y 580.798,Z 653.255,A -85,B 0,C 180,E1 -1787.752,E2 -1787.752} C_VEL
LIN {X 0,Y 580.74,Z 665.974,A -85,B 0,C 180,E1 -1788.039,E2 -1788.039} C_VEL
LIN {X 0,Y 580.637,Z 679.696,A -85,B 0,C 180,E1 -1788.515,E2 -1788.515} C_VEL
LIN {X 0,Y 580.556,Z 691.896,A -85,B 0,C 180,E1 -1789.097,E2 -1789.097} C_VEL
LIN {X 0,Y 580.449,Z 703.34,A -85,B 0,C 180,E1 -1789.8,E2 -1789.8} C_VEL
LIN {X 0,Y 580.37,Z 713.597,A -85,B 0,C 180,E1 -1790.591,E2 -1790.591} C_VEL
LIN {X 0,Y 580.28,Z 722.839,A -85,B 0,C 180,E1 -1791.468,E2 -1791.468} C_VEL
LIN {X 0,Y 580.221,Z 730.473,A -85,B 0,C 180,E1 -1792.343,E2 -1792.343} C_VEL
LIN {X 0,Y 580.17,Z 737.86,A -85,B 0,C 180,E1 -1793.377,E2 -1793.377} C_VEL
LIN {X 0,Y 580.139,Z 743.955,A -85,B 0,C 180,E1 -1794.438,E2 -1794.438} C_VEL
LIN {X 0,Y 580.107,Z 748.697,A -85,B 0,C 180,E1 -1795.483,E2 -1795.483} C_VEL
LIN {X 0,Y 580.123,Z 752.328,A -85,B 0,C 180,E1 -1796.527,E2 -1796.527} C_VEL
LIN {X 0,Y 580.043,Z 754.185,A -85,B 0,C 180,E1 -1797.222,E2 -1797.222} C_VEL
LIN {X 0,Y 580.047,Z 756.637,A -85,B 0,C 180,E1 -1798.611,E2 -1798.611} C_VEL
LIN {X 0,Y 580.041,Z 757.253,A -85,B 0,C 180,E1 -1799.306,E2 -1799.306} C_VEL
LIN {X 0,Y 580.04,Z 757.312,A -85,B 0,C 180,E1 -1800.694,E2 -1800.694} C_VEL
LIN {X 0,Y 580.047,Z 756.739,A -85,B 0,C 180,E1 -1801.389,E2 -1801.389} C_VEL
LIN {X 0,Y 580.044,Z 754.411,A -85,B 0,C 180,E1 -1802.778,E2 -1802.778} C_VEL
LIN {X 0,Y 580.109,Z 751.54,A -85,B 0,C 180,E1 -1803.821,E2 -1803.821} C_VEL
LIN {X 0,Y 580.054,Z 747.639,A -85,B 0,C 180,E1 -1804.865,E2 -1804.865} C_VEL
LIN {X 0,Y 580.161,Z 742.593,A -85,B 0,C 180,E1 -1805.91,E2 -1805.91} C_VEL
LIN {X 0,Y 580.157,Z 736.241,A -85,B 0,C 180,E1 -1806.958,E2 -1806.958} C_VEL
LIN {X 0,Y 580.241,Z 728.362,A -85,B 0,C 180,E1 -1808.007,E2 -1808.007} C_VEL
LIN {X 0,Y 580.308,Z 718.514,A -85,B 0,C 180,E1 -1809.058,E2 -1809.058} C_VEL
LIN {X 0,Y 580.407,Z 708.155,A -85,B 0,C 180,E1 -1809.936,E2 -1809.936} C_VEL
LIN {X 0,Y 580.503,Z 697.953,A -85,B 0,C 180,E1 -1810.639,E2 -1810.639} C_VEL
LIN {X 0,Y 580.594,Z 686.717,A -85,B 0,C 180,E1 -1811.261,E2 -1811.261} C_VEL
LIN {X 0,Y 580.66,Z 674.236,A -85,B 0,C 180,E1 -1811.785,E2 -1811.785} C_VEL
LIN {X 0,Y 580.776,Z 661.728,A -85,B 0,C 180,E1 -1812.16,E2 -1812.16} C_VEL
LIN {X 0,Y 580.836,Z 649.142,A -85,B 0,C 180,E1 -1812.402,E2 -1812.402} C_VEL
LIN {X 0,Y 580.867,Z 547.564,A -85,B 0,C 180,E1 -1813.668,E2 -1813.668} C_VEL
LIN {X 0,Y 580.438,Z 544.661,A -85,B 0,C 180,E1 -1813.724,E2 -1813.724} C_VEL
LIN {X 0,Y 580.604,Z 521.572,A -85,B 0,C 180,E1 -1816.707,E2 -1816.707} C_VEL
LIN {X 0,Y 580.803,Z 499.181,A -85,B 0,C 180,E1 -1819.643,E2 -1819.643} C_VEL
LIN {X 0,Y 581.035,Z 477.129,A -85,B 0,C 180,E1 -1822.584,E2 -1822.584} C_VEL
LIN {X 0,Y 581.128,Z 467.407,A -85,B 0,C 180,E1 -1823.9,E2 -1823.9} C_VEL
LIN {X 0,Y 580.318,Z 463.327,A -85,B 0,C 180,E1 -1824.505,E2 -1824.505} C_VEL
LIN {X 0,Y 580.285,Z 463.324,A -85,B 0,C 180,E1 -1827.402,E2 -1827.402} C_VEL
LIN {X 0,Y 580.291,Z 463.322,A -85,B 0,C 180,E1 -1829.773,E2 -1829.773} C_VEL
LIN {X 0,Y 580.3,Z 463.323,A -85,B 0,C 180,E1 -1832.201,E2 -1832.201} C_VEL
LIN {X 0,Y 580.294,Z 463.331,A -85,B 0,C 180,E1 -1834.696,E2 -1834.696} C_VEL
LIN {X 0,Y 580.3,Z 463.322,A -85,B 0,C 180,E1 -1837.268,E2 -1837.268} C_VEL
LIN {X 0,Y 580.298,Z 463.325,A -85,B 0,C 180,E1 -1840.271,E2 -1840.271} C_VEL
LIN {X 0,Y 580.278,Z 463.33,A -85,B 0,C 180,E1 -1842.706,E2 -1842.706} C_VEL
LIN {X 0,Y 580.277,Z 463.322,A -85,B 0,C 180,E1 -1845.608,E2 -1845.608} C_VEL
LIN {X 0,Y 580.317,Z 463.324,A -85,B 0,C 180,E1 -1848.234,E2 -1848.234} C_VEL
LIN {X 0,Y 580.281,Z 463.325,A -85,B 0,C 180,E1 -1850.965,E2 -1850.965} C_VEL
LIN {X 0,Y 580.295,Z 463.321,A -85,B 0,C 180,E1 -1853.598,E2 -1853.598} C_VEL
LIN {X 0,Y 580.307,Z 463.324,A -85,B 0,C 180,E1 -1856.683,E2 -1856.683} C_VEL
LIN {X 0,Y 580.313,Z 463.319,A -85,B 0,C 180,E1 -1859.426,E2 -1859.426} C_VEL
LIN {X 0,Y 580.301,Z 463.328,A -85,B 0,C 180,E1 -1862.141,E2 -1862.141} C_VEL
LIN {X 0,Y 580.325,Z 463.319,A -85,B 0,C 180,E1 -1865.269,E2 -1865.269} C_VEL
LIN {X 0,Y 580.346,Z 463.507,A -85,B 0,C 180,E1 -1866.467,E2 -1866.467} C_VEL
LIN {X 0,Y 581.231,Z 468.65,A -85,B 0,C 180,E1 -1867.111,E2 -1867.111} C_VEL
LIN {X 0,Y 581.001,Z 490.506,A -85,B 0,C 180,E1 -1869.649,E2 -1869.649} C_VEL
LIN {X 0,Y 580.766,Z 516.021,A -85,B 0,C 180,E1 -1872.564,E2 -1872.564} C_VEL
LIN {X 0,Y 580.689,Z 523.691,A -85,B 0,C 180,E1 -1873.431,E2 -1873.431} C_VEL
LIN {X 0,Y 581.396,Z 528.61,A -85,B 0,C 180,E1 -1873.519,E2 -1873.519} C_VEL
LIN {X 0,Y 581.127,Z 662.883,A -85,B 0,C 180,E1 -1875.22,E2 -1875.22} C_VEL
LIN {X 0,Y 581.059,Z 677.25,A -85,B 0,C 180,E1 -1875.55,E2 -1875.55} C_VEL
LIN {X 0,Y 580.907,Z 690.711,A -85,B 0,C 180,E1 -1875.997,E2 -1875.997} C_VEL
LIN {X 0,Y 580.8,Z 704.638,A -85,B 0,C 180,E1 -1876.619,E2 -1876.619} C_VEL
LIN {X 0,Y 580.656,Z 717.097,A -85,B 0,C 180,E1 -1877.328,E2 -1877.328} C_VEL
LIN {X 0,Y 580.526,Z 729.639,A -85,B 0,C 180,E1 -1878.212,E2 -1878.212} C_VEL
LIN {X 0,Y 580.441,Z 740.906,A -85,B 0,C 180,E1 -1879.19,E2 -1879.19} C_VEL
LIN {X 0,Y 580.275,Z 750.851,A -85,B 0,C 180,E1 -1880.238,E2 -1880.238} C_VEL
LIN {X 0,Y 580.241,Z 759.171,A -85,B 0,C 180,E1 -1881.292,E2 -1881.292} C_VEL
LIN {X 0,Y 580.166,Z 767.126,A -85,B 0,C 180,E1 -1882.518,E2 -1882.518} C_VEL
LIN {X 0,Y 580.102,Z 773.527,A -85,B 0,C 180,E1 -1883.74,E2 -1883.74} C_VEL
LIN {X 0,Y 580.078,Z 777.961,A -85,B 0,C 180,E1 -1884.787,E2 -1884.787} C_VEL
LIN {X 0,Y 580.102,Z 781.442,A -85,B 0,C 180,E1 -1885.831,E2 -1885.831} C_VEL
LIN {X 0,Y 580.041,Z 784.831,A -85,B 0,C 180,E1 -1887.222,E2 -1887.222} C_VEL
LIN {X 0,Y 580.041,Z 786.832,A -85,B 0,C 180,E1 -1888.611,E2 -1888.611} C_VEL
LIN {X 0,Y 580.036,Z 787.5,A -85,B 0,C 180,E1 -1890,E2 -1890} C_VEL
LIN {X 0,Y 580.041,Z 786.832,A -85,B 0,C 180,E1 -1891.389,E2 -1891.389} C_VEL
LIN {X 0,Y 580.041,Z 784.833,A -85,B 0,C 180,E1 -1892.778,E2 -1892.778} C_VEL
LIN {X 0,Y 580.102,Z 781.443,A -85,B 0,C 180,E1 -1894.169,E2 -1894.169} C_VEL
LIN {X 0,Y 580.128,Z 776.568,A -85,B 0,C 180,E1 -1895.562,E2 -1895.562} C_VEL
LIN {X 0,Y 580.141,Z 770.052,A -85,B 0,C 180,E1 -1896.958,E2 -1896.958} C_VEL
LIN {X 0,Y 580.192,Z 762.799,A -85,B 0,C 180,E1 -1898.183,E2 -1898.183} C_VEL
LIN {X 0,Y 580.284,Z 753.822,A -85,B 0,C 180,E1 -1899.41,E2 -1899.41} C_VEL
LIN {X 0,Y 580.356,Z 744.39,A -85,B 0,C 180,E1 -1900.466,E2 -1900.466} C_VEL
LIN {X 0,Y 580.476,Z 734.317,A -85,B 0,C 180,E1 -1901.404,E2 -1901.404} C_VEL
LIN {X 0,Y 580.597,Z 722.429,A -85,B 0,C 180,E1 -1902.319,E2 -1902.319} C_VEL
LIN {X 0,Y 580.73,Z 709.645,A -85,B 0,C 180,E1 -1903.115,E2 -1903.115} C_VEL
LIN {X 0,Y 580.911,Z 697.155,A -85,B 0,C 180,E1 -1903.735,E2 -1903.735} C_VEL
LIN {X 0,Y 581.019,Z 684.245,A -85,B 0,C 180,E1 -1904.234,E2 -1904.234} C_VEL
LIN {X 0,Y 581.082,Z 670.189,A -85,B 0,C 180,E1 -1904.631,E2 -1904.631} C_VEL
LIN {X 0,Y 581.164,Z 655.591,A -85,B 0,C 180,E1 -1904.891,E2 -1904.891} C_VEL
LIN {X 0,Y 581.352,Z 527.71,A -85,B 0,C 180,E1 -1906.493,E2 -1906.493} C_VEL
LIN {X 0,Y 580.688,Z 523.691,A -85,B 0,C 180,E1 -1906.569,E2 -1906.569} C_VEL
LIN {X 0,Y 580.927,Z 499.408,A -85,B 0,C 180,E1 -1909.328,E2 -1909.328} C_VEL
LIN {X 0,Y 581.188,Z 474.512,A -85,B 0,C 180,E1 -1912.203,E2 -1912.203} C_VEL
LIN {X 0,Y 581.213,Z 467.584,A -85,B 0,C 180,E1 -1913.015,E2 -1913.015} C_VEL
LIN {X 0,Y 580.311,Z 463.329,A -85,B 0,C 180,E1 -1913.557,E2 -1913.557} C_VEL
LIN {X 0,Y 580.296,Z 463.323,A -85,B 0,C 180,E1 -1916.334,E2 -1916.334} C_VEL
LIN {X 0,Y 580.304,Z 463.327,A -85,B 0,C 180,E1 -1919.31,E2 -1919.31} C_VEL
LIN {X 0,Y 580.305,Z 463.321,A -85,B 0,C 180,E1 -1922.2,E2 -1922.2} C_VEL
LIN {X 0,Y 580.29,Z 463.323,A -85,B 0,C 180,E1 -1924.696,E2 -1924.696} C_VEL
LIN {X 0,Y 580.302,Z 463.329,A -85,B 0,C 180,E1 -1927.269,E2 -1927.269} C_VEL
LIN {X 0,Y 580.293,Z 463.321,A -85,B 0,C 180,E1 -1930.271,E2 -1930.271} C_VEL
LIN {X 0,Y 580.285,Z 463.325,A -85,B 0,C 180,E1 -1932.706,E2 -1932.706} C_VEL
LIN {X 0,Y 580.261,Z 463.328,A -85,B 0,C 180,E1 -1935.61,E2 -1935.61} C_VEL
LIN {X 0,Y 580.282,Z 463.323,A -85,B 0,C 180,E1 -1938.231,E2 -1938.231} C_VEL
LIN {X 0,Y 580.294,Z 463.33,A -85,B 0,C 180,E1 -1940.966,E2 -1940.966} C_VEL
LIN {X 0,Y 580.273,Z 463.325,A -85,B 0,C 180,E1 -1943.597,E2 -1943.597} C_VEL
LIN {X 0,Y 580.322,Z 463.319,A -85,B 0,C 180,E1 -1946.146,E2 -1946.146} C_VEL
LIN {X 0,Y 580.292,Z 463.33,A -85,B 0,C 180,E1 -1948.615,E2 -1948.615} C_VEL
LIN {X 0,Y 580.297,Z 463.327,A -85,B 0,C 180,E1 -1951.024,E2 -1951.024} C_VEL
LIN {X 0,Y 580.296,Z 463.324,A -85,B 0,C 180,E1 -1953.666,E2 -1953.666} C_VEL
LIN {X 0,Y 580.304,Z 463.322,A -85,B 0,C 180,E1 -1955.684,E2 -1955.684} C_VEL
LIN {X 0,Y 580.298,Z 463.377,A -85,B 0,C 180,E1 -1956.834,E2 -1956.834} C_VEL
LIN {X 0,Y 581.104,Z 468.696,A -85,B 0,C 180,E1 -1957.606,E2 -1957.606} C_VEL
LIN {X 0,Y 580.864,Z 488.874,A -85,B 0,C 180,E1 -1960.356,E2 -1960.356} C_VEL
LIN {X 0,Y 580.665,Z 510.81,A -85,B 0,C 180,E1 -1963.294,E2 -1963.294} C_VEL
LIN {X 0,Y 580.514,Z 532.578,A -85,B 0,C 180,E1 -1966.166,E2 -1966.166} C_VEL
LIN {X 0,Y 580.409,Z 541.858,A -85,B 0,C 180,E1 -1967.378,E2 -1967.378} C_VEL
LIN {X 0,Y 580.971,Z 548.007,A -85,B 0,C 180,E1 -1967.468,E2 -1967.468} C_VEL
LIN {X 0,Y 580.799,Z 650.742,A -85,B 0,C 180,E1 -1968.758,E2 -1968.758} C_VEL
LIN {X 0,Y 580.756,Z 664.253,A -85,B 0,C 180,E1 -1969.078,E2 -1969.078} C_VEL
LIN {X 0,Y 580.593,Z 677.291,A -85,B 0,C 180,E1 -1969.539,E2 -1969.539} C_VEL
LIN {X 0,Y 580.524,Z 689.94,A -85,B 0,C 180,E1 -1970.154,E2 -1970.154} C_VEL
LIN {X 0,Y 580.441,Z 701.139,A -85,B 0,C 180,E1 -1970.856,E2 -1970.856} C_VEL
LIN {X 0,Y 580.371,Z 711.221,A -85,B 0,C 180,E1 -1971.645,E2 -1971.645} C_VEL
LIN {X 0,Y 580.253,Z 720.335,A -85,B 0,C 180,E1 -1972.519,E2 -1972.519} C_VEL
LIN {X 0,Y 580.203,Z 729.315,A -85,B 0,C 180,E1 -1973.578,E2 -1973.578} C_VEL
LIN {X 0,Y 580.124,Z 736.357,A -85,B 0,C 180,E1 -1974.613,E2 -1974.613} C_VEL
LIN {X 0,Y 580.107,Z 742.87,A -85,B 0,C 180,E1 -1975.831,E2 -1975.831} C_VEL
LIN {X 0,Y 580.093,Z 747.172,A -85,B 0,C 180,E1 -1976.875,E2 -1976.875} C_VEL
LIN {X 0,Y 580.049,Z 750.427,A -85,B 0,C 180,E1 -1977.917,E2 -1977.917} C_VEL
LIN {X 0,Y 580.048,Z 752.034,A -85,B 0,C 180,E1 -1978.611,E2 -1978.611} C_VEL
LIN {X 0,Y 580.04,Z 753.238,A -85,B 0,C 180,E1 -1979.306,E2 -1979.306} C_VEL
LIN {X 0,Y 580.039,Z 754.038,A -85,B 0,C 180,E1 -1980,E2 -1980} C_VEL
LIN {X 0,Y 580.047,Z 754.429,A -85,B 0,C 180,E1 -1981.389,E2 -1981.389} C_VEL
LIN {X 0,Y 580.037,Z 754.044,A -85,B 0,C 180,E1 -1982.083,E2 -1982.083} C_VEL
LIN {X 0,Y 580.04,Z 753.247,A -85,B 0,C 180,E1 -1982.778,E2 -1982.778} C_VEL
LIN {X 0,Y 580.109,Z 752.043,A -85,B 0,C 180,E1 -1983.473,E2 -1983.473} C_VEL
LIN {X 0,Y 580.102,Z 749.468,A -85,B 0,C 180,E1 -1984.517,E2 -1984.517} C_VEL
LIN {X 0,Y 580.126,Z 745.865,A -85,B 0,C 180,E1 -1985.562,E2 -1985.562} C_VEL
LIN {X 0,Y 580.125,Z 740.429,A -85,B 0,C 180,E1 -1986.753,E2 -1986.753} C_VEL
LIN {X 0,Y 580.165,Z 734.085,A -85,B 0,C 180,E1 -1987.833,E2 -1987.833} C_VEL
LIN {X 0,Y 580.225,Z 726.381,A -85,B 0,C 180,E1 -1988.884,E2 -1988.884} C_VEL
LIN {X 0,Y 580.291,Z 716.736,A -85,B 0,C 180,E1 -1989.938,E2 -1989.938} C_VEL
LIN {X 0,Y 580.406,Z 706.859,A -85,B 0,C 180,E1 -1990.808,E2 -1990.808} C_VEL
LIN {X 0,Y 580.461,Z 696.857,A -85,B 0,C 180,E1 -1991.523,E2 -1991.523} C_VEL
LIN {X 0,Y 580.594,Z 686.062,A -85,B 0,C 180,E1 -1992.141,E2 -1992.141} C_VEL
LIN {X 0,Y 580.664,Z 674.284,A -85,B 0,C 180,E1 -1992.672,E2 -1992.672} C_VEL
LIN {X 0,Y 580.717,Z 661.442,A -85,B 0,C 180,E1 -1993.093,E2 -1993.093} C_VEL
LIN {X 0,Y 580.816,Z 649.062,A -85,B 0,C 180,E1 -1993.358,E2 -1993.358} C_VEL
LIN {X 0,Y 580.86,Z 613.475,A -85,B 0,C 180,E1 -1993.811,E2 -1993.811} C_VEL
LIN {X 0,Y 580.204,Z 607.666,A -85,B 0,C 180,E1 -1993.898,E2 -1993.898} C_VEL
LIN {X 0,Y 574.672,Z 588.962,A -85,B 0,C 180,E1 -1994.258,E2 -1994.258} C_VEL
LIN {X 0,Y 574.047,Z 583.153,A -85,B 0,C 180,E1 -1994.346,E2 -1994.346} C_VEL
LIN {X 0,Y 573.883,Z 544.984,A -85,B 0,C 180,E1 -1994.831,E2 -1994.831} C_VEL
LIN {X 0,Y 573.394,Z 541.789,A -85,B 0,C 180,E1 -1994.891,E2 -1994.891} C_VEL
LIN {X 0,Y 573.661,Z 519.619,A -85,B 0,C 180,E1 -1997.835,E2 -1997.835} C_VEL
LIN {X 0,Y 573.851,Z 497.607,A -85,B 0,C 180,E1 -2000.804,E2 -2000.804} C_VEL
LIN {X 0,Y 574.131,Z 477.742,A -85,B 0,C 180,E1 -2003.524,E2 -2003.524} C_VEL
LIN {X 0,Y 574.054,Z 468.083,A -85,B 0,C 180,E1 -2004.875,E2 -2004.875} C_VEL
LIN {X 0,Y 573.27,Z 464.2,A -85,B 0,C 180,E1 -2005.458,E2 -2005.458} C_VEL
LIN {X 0,Y 573.25,Z 464.203,A -85,B 0,C 180,E1 -2008.028,E2 -2008.028} C_VEL
LIN {X 0,Y 573.249,Z 464.201,A -85,B 0,C 180,E1 -2010.176,E2 -2010.176} C_VEL
